(* PLC project ArfBot.project, CODESYS CODESYS V3.5 SP19 Patch 4 *)
(* stored: creationDateTime 2024-02-26T21:29:06.3801046, modificationDateTime 2024-02-26T21:28:27.7609543 *)

TYPE ST_CncCmd :
STRUCT
	StartPos: 		SMC_PosInfo;				
	OriConvention: 	SMC_ORI_CONVENTION:=SMC_ORI_CONVENTION.ZYX;
	Filename: 		STRING:='CNC_FromFile.cnc';
	CoordinateType: DUT_Command_CoordinateType:=DUT_Command_CoordinateType.Variable;
	ArrayIndex: 	INT:=GVL.DEC_START_POS;
	ArrayType: 		DUT_Command_ArrayType:=DUT_Command_ArrayType.StoredPosition;
END_STRUCT
END_TYPE

TYPE DUT_Command :
STRUCT
	CommandType: DUT_CommandType;
	CommandString: STRING(GVL.COMMAND_LEN);
END_STRUCT
END_TYPE

TYPE DUT_Program :
STRUCT
	ProgramName: STRING;
	Commands: ARRAY [GVL.PROG_CMDS_ARR_BEG..GVL.PROG_CMDS_ARR_END] OF DUT_Command;
END_STRUCT
END_TYPE

TYPE DUT_StoredPosition :
STRUCT
	Comment: STRING;
	Position: MC_COORD_REF;
END_STRUCT
END_TYPE

TYPE ST_VisionLocate :
STRUCT
    MaxParts: 		UINT:=1; // max number of parts to locate
    MaxOverlap: 	REAL:=0.0; // max overlap of parts. only needed if MaxParts is greater than zero.
    Score: 			REAL:=0.6; // min score
    ToleranceAngle: REAL:=90.0; // max angle +/- to search
	ResultPosition: UINT:=0; // location to store the results in the vision register array
	TemplateName: 	STRING:='Template.jpg'; // name of the template to search
	ScriptFilename: STRING:='FastTemplateMatching.py'; // name of the script that runs the vision program
END_STRUCT
END_TYPE

TYPE ST_VisionCalibrate :
STRUCT
    CheckerSize: REAL:=25.0; // this value is in user units ex mm
    CheckerXCount: UINT:=6; // count of checker blocks in x coordinate
    CheckerYCount: UINT:=9; // count of checker blocks in y coordinate
END_STRUCT
END_TYPE

TYPE ST_VisionCmd :
STRUCT
    CommandType: DUT_Command_VisionType;
    ImageWidth: UINT:=640; // pixel count in x direction (must be supported by camera)
    ImageHeight: UINT:=400; // pixel coutn in y direction (must be supported by camera)
    Calibrate: ST_VisionCalibrate;
    Locate: ST_VisionLocate;
	Timeout: UDINT:=60; // timeout in seconds
END_STRUCT
END_TYPE

TYPE DUT_VisionRegister EXTENDS DUT_StoredPosition :
STRUCT
	Scaling: REAL;
END_STRUCT
END_TYPE

TYPE DUT_Flags :
STRUCT
	Comment: STRING:='';
	Value: BOOL:=FALSE;
END_STRUCT
END_TYPE

TYPE ST_MoveCmd :
STRUCT
	// common
	MoveType: 					DUT_Command_MoveType:=DUT_Command_MoveType.DirectMove;
	Speed: 						LREAL:=0.0;
	CoordSystem: 				SMC_COORD_SYSTEM:=SMC_COORD_SYSTEM.ACS;
	
	// direct/linear moves
	PositionType: 				DUT_Command_PositionType:=DUT_Command_PositionType.AbsolutePosition;
	CoordinateType: 			DUT_Command_CoordinateType:=DUT_Command_CoordinateType.Literal;
	ArrayIndex: 				UINT:=0;
	ArrayType: 					DUT_Command_ArrayType:=DUT_Command_ArrayType.StoredPosition;
	CoordRef: 					MC_COORD_REF:=(X:=0, Y:=0, Z:=0, A:=0, B:=0, C:=0);
	
	// circular moves
	CircularCoordinateType: 	DUT_Command_CoordinateType:=DUT_Command_CoordinateType.Literal;
	CircularArrayIndex: 		UINT:=0;
	CircularArrayType: 			DUT_Command_ArrayType:=DUT_Command_ArrayType.StoredPosition;
	CircleMode: 				SMC_CIRC_MODE:=SMC_CIRC_MODE.CENTER;
	PathChoice: 				MC_CIRC_PATHCHOICE:=MC_CIRC_PATHCHOICE.CLOCKWISE;
	CoordRef2: 					MC_COORD_REF:=(X:=0, Y:=0, Z:=0, A:=0, B:=0, C:=0);
	
END_STRUCT
END_TYPE

TYPE ST_OutputCmd :
STRUCT
	OutputType: DUT_OutputType;
	OutputTarget: INT;
	OutputValue1: LREAL;
	OutputValue2: LREAL;
END_STRUCT
END_TYPE

TYPE ST_PauseCmd :
STRUCT
	PauseTime: TIME:=T#1S;
END_STRUCT
END_TYPE

TYPE ST_VarSetCmd :
STRUCT
	ArrayType: DUT_Command_ArrayType;
	ArrayIndex: INT;
	Coordinates: MC_COORD_REF;
END_STRUCT
END_TYPE

TYPE ST_LogicCmdIO :
STRUCT
	Input: ARRAY [GVL.DIG_IN_ARR_BEG..GVL.DIG_IN_ARR_END] OF BOOL;
	Output: ARRAY [GVL.DIG_OUT_ARR_BEG..GVL.DIG_OUT_ARR_END] OF BOOL;
	Register: ARRAY [GVL.REG_ARR_BEG..GVL.REG_ARR_END] OF UDINT;
	Counter: ARRAY [GVL.REG_ARR_BEG..GVL.REG_ARR_END] OF UDINT;
END_STRUCT
END_TYPE

TYPE ST_LogicCmd :
STRUCT
	IF_Condition : E_LogicIfCondition;
	IF_Condition_Idx: INT;
	IF_Condition_Operator: E_LogicIfConditionOperator;
	IF_Condition_Operator_Value: UDINT;
	THEN_Function: E_LogicFunction;
	THEN_Function_Value: UDINT;
	THEN_Function_Idx: INT;
	ELSE_Function: E_LogicFunction;
	ELSE_Function_Idx: INT;
	ELSE_Function_Value: UDINT;
END_STRUCT
END_TYPE

INTERFACE ITFModule
METHOD M_Start
VAR_INPUT
END_VAR
END_METHOD
METHOD M_Stop
VAR_INPUT
END_VAR
END_METHOD
METHOD M_Home
VAR_INPUT
END_VAR
END_METHOD
METHOD M_Abort
VAR_INPUT
END_VAR
END_METHOD
METHOD M_Hold
VAR_INPUT
END_VAR
END_METHOD
{attribute 'monitoring' := 'variable'}
PROPERTY PropCurrentState : PACK_ML.State
END_PROPERTY
{attribute 'monitoring' := 'variable'}
PROPERTY PropBusy : BOOL
END_PROPERTY
{attribute 'monitoring' := 'variable'}
PROPERTY PropError : BOOL
END_PROPERTY
{attribute 'monitoring' := 'variable'}
PROPERTY PropErrDescription : STRING
END_PROPERTY
END_INTERFACE

TYPE StringByteArray : UNION
  bArray : ARRAY[0..254] OF BYTE;
  sString : STRING(255);
END_UNION;
END_TYPE

PROGRAM _00_Main
VAR
	// drive parameters
	//SM_Drive_PosControl_J1.controller.fDeadTime := 2.0;
	//SM_Drive_PosControl_J2.controller.fDeadTime := 2.0;
	//SM_Drive_PosControl_J3.controller.fDeadTime := 2.0;
	//SM_Drive_PosControl_J4.controller.fDeadTime := 2.0;
	//SM_Drive_PosControl_J5.controller.fDeadTime := 2.0;
	//SM_Drive_PosControl_J6.controller.fDeadTime := 2.0;
	
	// homing
	SMC_Homing_J1,SMC_Homing_J2,SMC_Homing_J3: SMC_Homing;
	SMC_Homing_J4,SMC_Homing_J5,SMC_Homing_J6: SMC_Homing;
	HomingSequence: INT := 0;
	SMC_GroupPower_J: SMC_GroupPower;
	MC_GroupReset_J: MC_GroupReset;
	MC_GroupEnable_J : MC_GroupEnable;
	MC_GroupDisable_J : MC_GroupDisable;
	HomingVelocityFast: LREAL:= 20.0;
	HomingAcceleration: LREAL:= 100.0;
	
	// jogging
	ProcessJog: JogProcessor;
	JogStatusText: STRING(255);
	
	// cnc
	VisuStruct3DControl_J: VisuStruct3DControl;
	TrackPosition: PositionTracker;
	
	// command processor
	PowerOn: BOOL:=FALSE;
	_MoveCommandParser: ParseMoveCmd;
	ProcessMoveCommand: MoveCmdProcessor;
	ProcessMoveCommand_Execute: BOOL;
	ProcessMoveCommand_Reset: BOOL;
	ProcessMoveStatusText: STRING(255);
	ProcessCommands: CommandProcessor;
	ProcessCommands_Execute: BOOL;
	ProcessCommand_Cancel: BOOL;
	ProcessCommand_Reset: BOOL;
	ProcessCommand_ActiveProgram: UINT := 0;
	StMoveCmdPose1: ST_MoveCmd;
	StMoveCmdPose2: ST_MoveCmd;
	Abort: BOOL;
	
	// vision
	Vision_pResultRtrig: R_TRIG;
	Vision_BitmapVersion: INT;
	Vision_CaptureImage: BOOL;
	Vision_CapImgCmdAccepted: BOOL;
	Vision_RunCalibration: BOOL;
	Vision_RunCalCmdAccepted: BOOL;
	Vision_LocatePart: BOOL;
	Vision_LocPartCmdAccepted: BOOL;
	Vision_StreamCamera: BOOL;
	Vision_StrCamCmdAccepted: BOOL;
	Vision_Cancel: BOOL;
	Vision_Reset: BOOL;
	
	//
	BuildTests: BOOL:=FALSE;
	FirstScan: BOOL:=TRUE;

END_VAR

                    
{region "utility"}
		 
	IF FirstScan THEN
		A_Init();	
	END_IF
	
	IF BuildTests THEN
		BuildTests := FALSE;
		M_BuildTests();
	END_IF
	
{endregion}
     
{region "methods"}

    A_Jogging();
    A_Homing();
    A_CNC();
    A_Processor();
    A_Vision();
    
{endregion}

FirstScan:=FALSE;
                  

ACTION A_Homing:
                        IF NOT GVL.PowerOn AND HomingSequence > 0 AND HomingSequence < 999  THEN
	HomingSequence := 999;
END_IF

CASE HomingSequence OF
  999: //
		SMC_GroupPower_J.Enable := FALSE;
		SMC_GroupPower_J.bDriveStart := FALSE;
		SMC_GroupPower_J.bRegulatorOn := FALSE;
		MC_GroupEnable_J.Execute := FALSE;
		MC_GroupDisable_J.Execute := FALSE;
		ProcessMoveCommand_Execute := FALSE;
		SMC_Homing_J1.bExecute := FALSE;
		SMC_Homing_J2.bExecute := FALSE;
		SMC_Homing_J3.bExecute := FALSE;
		SMC_Homing_J4.bExecute := FALSE;
		SMC_Homing_J5.bExecute := FALSE;
		SMC_Homing_J6.bExecute := FALSE;
		SM_Drive_PosControl_J1.bSWLimitEnable := TRUE;
		SM_Drive_PosControl_J2.bSWLimitEnable := TRUE;
		SM_Drive_PosControl_J3.bSWLimitEnable := TRUE;
		SM_Drive_PosControl_J4.bSWLimitEnable := TRUE;
		SM_Drive_PosControl_J5.bSWLimitEnable := TRUE;
		SM_Drive_PosControl_J6.bSWLimitEnable := TRUE;
  		HomingSequence := 0;
		
	0: //
		IF GVL.Homing AND GVL.PowerOn THEN
			GVL.Homing := FALSE;
			SMC_GroupPower_J.Enable := TRUE;
			SMC_GroupPower_J.bDriveStart := TRUE;
			SMC_GroupPower_J.bRegulatorOn := TRUE;
			PersistentVars.Flags[GVL.HOME_COMPLETE].Value := FALSE;
			HomingSequence := 5;
		END_IF
		
	5:
		IF SMC_GroupPower_J.Status THEN
			MC_GroupEnable_J.Execute := TRUE;
			HomingSequence := 10;
		END_IF
		
	10:
		IF NOT MC_GroupEnable_J.Busy THEN
			HomingSequence := 20;
		END_IF
		
	20: //
		SMC_Homing_J1.bExecute := TRUE;
		SMC_Homing_J2.bExecute := TRUE;
		SMC_Homing_J3.bExecute := TRUE;
		SMC_Homing_J4.bExecute := TRUE;
		SMC_Homing_J5.bExecute := TRUE;
		SMC_Homing_J6.bExecute := TRUE;
		SMC_Homing_J1.bReturnToZero := FALSE;
		SMC_Homing_J2.bReturnToZero := FALSE;
		SMC_Homing_J3.bReturnToZero := FALSE;
		SMC_Homing_J4.bReturnToZero := FALSE;
		SMC_Homing_J5.bReturnToZero := FALSE;
		SMC_Homing_J6.bReturnToZero := FALSE;
		SMC_Homing_J1.fVelocitySlow := 10.0;
		SMC_Homing_J2.fVelocitySlow := 10.0;
		SMC_Homing_J3.fVelocitySlow := 10.0;
		SMC_Homing_J4.fVelocitySlow := 10.0;
		SMC_Homing_J5.fVelocitySlow := 10.0;
		SMC_Homing_J6.fVelocitySlow := 10.0;
		SM_Drive_PosControl_J1.bSWLimitEnable := FALSE;
		SM_Drive_PosControl_J2.bSWLimitEnable := FALSE;
		SM_Drive_PosControl_J3.bSWLimitEnable := FALSE;
		SM_Drive_PosControl_J4.bSWLimitEnable := FALSE;
		SM_Drive_PosControl_J5.bSWLimitEnable := FALSE;
		SM_Drive_PosControl_J6.bSWLimitEnable := FALSE;
		HomingSequence := 30;
		
	30: //
		IF SMC_Homing_J1.bDone
			AND SMC_Homing_J2.bDone
			AND SMC_Homing_J3.bDone
			AND SMC_Homing_J4.bDone
			AND SMC_Homing_J5.bDone
			AND SMC_Homing_J6.bDone THEN
				SMC_Homing_J1.bExecute := FALSE;
				SMC_Homing_J2.bExecute := FALSE;
				SMC_Homing_J3.bExecute := FALSE;
				SMC_Homing_J4.bExecute := FALSE;
				SMC_Homing_J5.bExecute := FALSE;
				SMC_Homing_J6.bExecute := FALSE;
				HomingSequence := 40;
		END_IF
		
	40: //
		SMC_Homing_J1.bExecute := TRUE;
		SMC_Homing_J2.bExecute := TRUE;
		SMC_Homing_J3.bExecute := TRUE;
		SMC_Homing_J4.bExecute := TRUE;
		SMC_Homing_J5.bExecute := TRUE;
		SMC_Homing_J6.bExecute := TRUE;
		IF NOT PersistentVars.Flags[GVL.HOM_TO_POSE_IDX].Value THEN
			SMC_Homing_J1.bReturnToZero := TRUE;
			SMC_Homing_J2.bReturnToZero := TRUE;
			SMC_Homing_J3.bReturnToZero := TRUE;
			SMC_Homing_J4.bReturnToZero := TRUE;
			SMC_Homing_J5.bReturnToZero := TRUE;
			SMC_Homing_J6.bReturnToZero := TRUE;
		END_IF
		SMC_Homing_J1.fVelocitySlow := 2.0;
		SMC_Homing_J2.fVelocitySlow := 2.0;
		SMC_Homing_J3.fVelocitySlow := 2.0;
		SMC_Homing_J4.fVelocitySlow := 2.0;
		SMC_Homing_J5.fVelocitySlow := 2.0;
		SMC_Homing_J6.fVelocitySlow := 2.0;
		HomingSequence := 50;
		
	50: //
		IF SMC_Homing_J1.bDone
			AND SMC_Homing_J2.bDone
			AND SMC_Homing_J3.bDone
			AND SMC_Homing_J4.bDone
			AND SMC_Homing_J5.bDone
			AND SMC_Homing_J6.bDone THEN
				SMC_Homing_J1.bExecute := FALSE;
				SMC_Homing_J2.bExecute := FALSE;
				SMC_Homing_J3.bExecute := FALSE;
				SMC_Homing_J4.bExecute := FALSE;
				SMC_Homing_J5.bExecute := FALSE;
				SMC_Homing_J6.bExecute := FALSE;
				IF NOT PersistentVars.Flags[GVL.HOM_TO_POSE_IDX].Value THEN
					HomingSequence := 60;
				ELSE
					HomingSequence := 100;
				END_IF
				PersistentVars.Flags[GVL.HOME_COMPLETE].Value := TRUE;
		END_IF
		
	60:
		MC_GroupDisable_J.Execute := TRUE;
		HomingSequence := 70;
		
	70:
		IF NOT MC_GroupDisable_J.Busy THEN
			HomingSequence := 999;
		END_IF
		
	100: //
		ProcessMoveCommand.Command := GVL.Pose2;
		ProcessMoveCommand.M_Start();
		HomingSequence := 110;
		
	110: //
		IF ProcessMoveCommand.ItfUnitMode.CurrentState = PACK_ML.State.Idle 
			OR NOT ProcessMoveCommand_Execute THEN
				ProcessMoveCommand_Execute := FALSE;
				HomingSequence := 999;
		END_IF

END_CASE

SMC_Homing_J1(
	Axis:=SM_Drive_PosControl_J1 , 
	bExecute:= ,
	fHomePosition:= PersistentVars.StoredPositions[GVL.HOM_POS_IDX].Position.X, 
	fVelocitySlow:= , 
	fVelocityFast:= HomingVelocityFast, 
	fAcceleration:= HomingAcceleration, 
	fDeceleration:= HomingAcceleration, 
	fJerk:= 1000.0, 
	nDirection:= MC_direction.negative, 
	bReferenceSwitch:= NOT _10_Drives.rx_j1_limit, 
	fSignalDelay:= , 
	nHomingMode:= , 
	bReturnToZero:= , 
	bIndexOccured:= , 
	fIndexPosition:= , 
	bIgnoreHWLimit:= TRUE, 
	bDone=> , 
	bBusy=> , 
	bCommandAborted=> , 
	bError=> , 
	nErrorID=> , 
	bStartLatchingIndex=> );
	
SMC_Homing_J2(
	Axis:=SM_Drive_PosControl_J2 , 
	bExecute:= , 
	fHomePosition:= PersistentVars.StoredPositions[GVL.HOM_POS_IDX].Position.Y,  
	fVelocitySlow:= , 
	fVelocityFast:= HomingVelocityFast, 
	fAcceleration:= HomingAcceleration, 
	fDeceleration:= HomingAcceleration,
	fJerk:= 1000.0, 
	nDirection:= MC_Direction.negative, 
	bReferenceSwitch:= NOT _10_Drives.rx_j2_limit, 
	fSignalDelay:= , 
	nHomingMode:= , 
	bReturnToZero:= , 
	bIndexOccured:= , 
	fIndexPosition:= , 
	bIgnoreHWLimit:= TRUE, 
	bDone=> , 
	bBusy=> , 
	bCommandAborted=> , 
	bError=> , 
	nErrorID=> , 
	bStartLatchingIndex=> );
	
SMC_Homing_J3(
	Axis:=SM_Drive_PosControl_J3 , 
	bExecute:= , 
	fHomePosition:= PersistentVars.StoredPositions[GVL.HOM_POS_IDX].Position.Z, 
	fVelocitySlow:= , 
	fVelocityFast:= HomingVelocityFast, 
	fAcceleration:= HomingAcceleration, 
	fDeceleration:= HomingAcceleration,
	fJerk:= 1000.0, 
	nDirection:= MC_Direction.positive, 
	bReferenceSwitch:= NOT _10_Drives.rx_j3_limit, 
	fSignalDelay:= , 
	nHomingMode:= , 
	bReturnToZero:= , 
	bIndexOccured:= , 
	fIndexPosition:= , 
	bIgnoreHWLimit:= TRUE, 
	bDone=> , 
	bBusy=> , 
	bCommandAborted=> , 
	bError=> , 
	nErrorID=> , 
	bStartLatchingIndex=> );
	
SMC_Homing_J4(
	Axis:=SM_Drive_PosControl_J4 , 
	bExecute:= ,
	fHomePosition:= PersistentVars.StoredPositions[GVL.HOM_POS_IDX].Position.A, 
	fVelocitySlow:= , 
	fVelocityFast:= HomingVelocityFast, 
	fAcceleration:= HomingAcceleration, 
	fDeceleration:= HomingAcceleration,
	fJerk:= 1000.0, 
	nDirection:= MC_Direction.positive, 
	bReferenceSwitch:= NOT _10_Drives.rx_j4_limit, 
	fSignalDelay:= , 
	nHomingMode:= , 
	bReturnToZero:= , 
	bIndexOccured:= , 
	fIndexPosition:= , 
	bIgnoreHWLimit:= TRUE, 
	bDone=> , 
	bBusy=> , 
	bCommandAborted=> , 
	bError=> , 
	nErrorID=> , 
	bStartLatchingIndex=> );
	
SMC_Homing_J5(
	Axis:=SM_Drive_PosControl_J5 , 
	bExecute:= , 
	fHomePosition:= PersistentVars.StoredPositions[GVL.HOM_POS_IDX].Position.B,  
	fVelocitySlow:= , 
	fVelocityFast:= HomingVelocityFast, 
	fAcceleration:= HomingAcceleration, 
	fDeceleration:= HomingAcceleration,
	fJerk:= 1000, 
	nDirection:= MC_Direction.positive, 
	bReferenceSwitch:= NOT _10_Drives.rx_j5_limit, 
	fSignalDelay:= , 
	nHomingMode:= , 
	bReturnToZero:= , 
	bIndexOccured:= , 
	fIndexPosition:= , 
	bIgnoreHWLimit:= TRUE, 
	bDone=> , 
	bBusy=> , 
	bCommandAborted=> , 
	bError=> , 
	nErrorID=> , 
	bStartLatchingIndex=> );
	
SMC_Homing_J6(
	Axis:=SM_Drive_PosControl_J6 , 
	bExecute:= , 
	fHomePosition:= PersistentVars.StoredPositions[GVL.HOM_POS_IDX].Position.C, 
	fVelocitySlow:= , 
	fVelocityFast:= HomingVelocityFast, 
	fAcceleration:= HomingAcceleration, 
	fDeceleration:= HomingAcceleration,
	fJerk:= 1000.0, 
	nDirection:= MC_Direction.negative, 
	bReferenceSwitch:= NOT _10_Drives.rx_j6_limit, 
	fSignalDelay:= , 
	nHomingMode:= , 
	bReturnToZero:= , 
	bIndexOccured:= , 
	fIndexPosition:= , 
	bIgnoreHWLimit:= TRUE, 
	bDone=> , 
	bBusy=> , 
	bCommandAborted=> , 
	bError=> , 
	nErrorID=> , 
	bStartLatchingIndex=> );

SMC_GroupPower_J(
	AxisGroup:= ArfBotAxisGroup, 
	Enable:=,
	bRegulatorOn:= SMC_GroupPower_J.Enable,
	bDriveStart:= SMC_GroupPower_J.Enable, 
	Status=> , 
	Busy=> , 
	Error=> , 
	ErrorID=> );
		 
MC_GroupEnable_J(
	AxisGroup:=ArfBotAxisGroup,
	Execute:=,
	CompatibilityOptions:=,
	Done=>,
	Busy=>,
	Error=>,
	ErrorID=>);
		 
MC_GroupDisable_J(
	AxisGroup:=ArfBotAxisGroup,
	Execute:=,
	Done=>,
	Busy=>,
	Error=>,
	ErrorID=>);	
		 
MC_GroupReset_J(
	AxisGroup:=ArfBotAxisGroup , 
	Execute:= GVL.Reset, 
	Done=> , 
	Busy=> , 
	Error=> , 
	ErrorID=> );
                      
END_ACTION

ACTION A_Processor:
                        
//	TODO need to get this removed and instead build a program for the poses
IF GVL.MoveToPose1 THEN
	GVL.MoveToPose1 := FALSE;
	IF GVL.PowerOn AND PersistentVars.Flags[GVL.HOME_COMPLETE].Value THEN
		ProcessMoveCommand.Command := GVL.Pose1;
		ProcessMoveCommand.M_Start();
	END_IF
ELSIF GVL.MoveToPose2 THEN
	GVL.MoveToPose2 := FALSE;
	IF GVL.PowerOn AND PersistentVars.Flags[GVL.HOME_COMPLETE].Value THEN
		ProcessMoveCommand.Command := GVL.Pose2;
		ProcessMoveCommand.M_Start();
	END_IF
END_IF

// TODO need to get this removed and instead build a program for the poses
ProcessMoveCommand(
	StoredPositions:= PersistentVars.StoredPositions,
	VisionRegisters:= PersistentVars.VisionRegisters,
	Flags:= PersistentVars.Flags,
	AxisGroup:= ArfBotAxisGroup, 
	Acceleration:= 1000, 
	AccFactor:= 0.05,
	Jerk:= 1000,
	JerkFactor:= 1, 
	Position=> ,
	ItfUnitMode=> , 
	Error=> );
IF ProcessMoveCommand_Reset OR GVL.Reset THEN
	ProcessMoveCommand_Reset := FALSE;
	ProcessMoveStatusText := '';
	ProcessMoveCommand.M_Home();
END_IF
IF ProcessMoveCommand.Error THEN
	ProcessMoveStatusText := CONCAT('Move Processor Error: ',ProcessMoveCommand.ErrorDescription) ;
END_IF

//
IF Abort THEN
	Abort := FALSE;
	IF NOT GVL.PowerOn THEN
		ProcessCommands.M_Abort();
		ProcessMoveCommand.M_Abort();
	END_IF
END_IF
IF ProcessCommands_Execute THEN
	ProcessCommands_Execute := FALSE;
	ProcessCommands.Commands := PersistentVars.Programs[ProcessCommand_ActiveProgram].Commands;
	ProcessCommands.M_Start();
END_IF
IF ProcessCommand_Cancel THEN
	ProcessCommand_Cancel := FALSE;
	ProcessCommands.M_Stop();
END_IF
IF ProcessCommand_Reset OR GVL.Reset THEN
	ProcessCommand_Reset := FALSE;
	ProcessCommands.M_Home();
END_IF
ProcessCommands(
	StoredPositions:=PersistentVars.StoredPositions,
	VisionRegisters:=PersistentVars.VisionRegisters,
	Flags:=PersistentVars.Flags,
	AxisGroup:= ArfBotAxisGroup,
	Servo1:= AdafruitPwm01,
	Servo2:= AdafruitPwm02,
	Enable:= GVL.PowerOn AND PersistentVars.Flags[GVL.HOME_COMPLETE].Value,
	Commands:= , 
	ActiveCommand => ,
	Error=> ,
	StatusText=>);	
                      
END_ACTION

ACTION A_CNC:
                        
// track position of robot end effector to display on hmi
TrackPosition(
	AxisGroup:=ArfBotAxisGroup,
	SM3_Drive_PosControl_J1:=SM_Drive_PosControl_J1,
	SM3_Drive_PosControl_J2:=SM_Drive_PosControl_J2,
	SM3_Drive_PosControl_J3:=SM_Drive_PosControl_J3,
	SM3_Drive_PosControl_J4:=SM_Drive_PosControl_J4,
	SM3_Drive_PosControl_J5:=SM_Drive_PosControl_J5,
	SM3_Drive_PosControl_J6:=SM_Drive_PosControl_J6,
	VisuStruct3DTrack=>,
	Arm=>,
	Elbow=>,
	Hand=>);
	
(*ProcessCnc(
	AxisGroup:=ArfBotAxisGroup,
	SM3_Drive_PosControl_J1:=SM_Drive_PosControl_J1,
	SM3_Drive_PosControl_J2:=SM_Drive_PosControl_J2,
	SM3_Drive_PosControl_J3:=SM_Drive_PosControl_J3,
	SM3_Drive_PosControl_J4:=SM_Drive_PosControl_J4,
	SM3_Drive_PosControl_J5:=SM_Drive_PosControl_J5,
	SM3_Drive_PosControl_J6:=SM_Drive_PosControl_J6,
	GapVelocity:= , 
	AvoidGaps:= , 
	GapAccel:= );*)

// set the start position for the MC_NCDecoder
// alternatively, we can set this in the CNC program properties
(*GVL.StartPos.dX:=PersistentVars.StoredPositions[GVL.DEC_START_POS].Position.X;
GVL.StartPos.dY:=PersistentVars.StoredPositions[GVL.DEC_START_POS].Position.Y;
GVL.StartPos.dZ:=PersistentVars.StoredPositions[GVL.DEC_START_POS].Position.Z;
GVL.StartPos.dA:=PersistentVars.StoredPositions[GVL.DEC_START_POS].Position.A;
GVL.StartPos.dB:=PersistentVars.StoredPositions[GVL.DEC_START_POS].Position.B;
GVL.StartPos.dC:=PersistentVars.StoredPositions[GVL.DEC_START_POS].Position.C;

IF TestExecute THEN
	TestExecute := FALSE;
	ProcessCnc.M_Execute(	FileName:='CNC_FromFile.cnc', 
							StartPos:=GVL.StartPos); // TODO 
END_IF
IF TestReset THEN
	TestReset := FALSE;
	ProcessCnc.M_Reset();
END_IF
IF TestCancel THEN
	TestCancel := FALSE;
	ProcessCnc.M_Cancel();
END_IF*)
                      
END_ACTION

ACTION A_Jogging:
                        
ProcessJog(
	AxisGroup:= ArfBotAxisGroup,
	Enable:= GVL.PowerOn,
	Reset:= GVL.Reset,
	ABC_as_ACS=>,
	CoordSystem=>, 
	Position=>, 
	Done=> , 
	Busy=> , 
	Error=> , 
	ErrorID=> );
IF ProcessJog.Reset THEN
	JogStatusText := '';
END_IF
IF ProcessJog.Error THEN
	JogStatusText := CONCAT('Jog Processor Error: ',
						CONCAT(TO_STRING(ProcessJog.ErrorID),
						CONCAT(' ', SMC_ErrorString(ProcessJog.ErrorID,
									SMC_Language_Type.english)))) ;
END_IF

                      
END_ACTION

ACTION A_Vision:
                        
// tell HMI to update image
//Vision_pResultRtrig(clk := _40_Vision.ProcessVisionCommand.ItfUnitMode.CurrentState = PACK_ML.State.Idle); TODO this causes an exception because ProcessVisionCommand has not went through first scan yet
Vision_pResultRtrig(clk := NOT _40_Vision.ProcessVisionCommand.Busy);
IF Vision_pResultRtrig.Q THEN
	Vision_BitmapVersion := Vision_BitmapVersion + 1;
END_IF

                      
END_ACTION

ACTION A_Init:
                        
// check if arfbot has been initialized
IF NOT PersistentVars.Flags[GVL.INIT_POS_IDX].Value THEN
	// poses
	PersistentVars.Flags[GVL.HOM_TO_POSE_IDX].Value := FALSE;
	PersistentVars.StoredPositions[GVL.POSE_1_IDX].Position.X := 0.0;
	PersistentVars.StoredPositions[GVL.POSE_1_IDX].Position.Y := 0.0;
	PersistentVars.StoredPositions[GVL.POSE_1_IDX].Position.Z := -30.0;
	PersistentVars.StoredPositions[GVL.POSE_1_IDX].Position.A := 0.0;
	PersistentVars.StoredPositions[GVL.POSE_1_IDX].Position.B := -30.0;
	PersistentVars.StoredPositions[GVL.POSE_1_IDX].Position.C := 0.0;
	PersistentVars.StoredPositions[GVL.POSE_2_IDX].Position.X := 0.0;
	PersistentVars.StoredPositions[GVL.POSE_2_IDX].Position.Y := 30.0;
	PersistentVars.StoredPositions[GVL.POSE_2_IDX].Position.Z := -30.0;
	PersistentVars.StoredPositions[GVL.POSE_2_IDX].Position.A := 0.0;
	PersistentVars.StoredPositions[GVL.POSE_2_IDX].Position.B := 30.0;
	PersistentVars.StoredPositions[GVL.POSE_2_IDX].Position.C := 0.0;
		 
	// decoder
	PersistentVars.StoredPositions[GVL.DEC_START_POS].Position.X := 300.0; // TODO need to verify all 6 of these
	PersistentVars.StoredPositions[GVL.DEC_START_POS].Position.Y := 0.0;
	PersistentVars.StoredPositions[GVL.DEC_START_POS].Position.Z := -400.0;
	PersistentVars.StoredPositions[GVL.DEC_START_POS].Position.A := 0.0;
	PersistentVars.StoredPositions[GVL.DEC_START_POS].Position.B := 0.0;
	PersistentVars.StoredPositions[GVL.DEC_START_POS].Position.C := 0.0;
		 
	
	// set homing offsets
	PersistentVars.StoredPositions[GVL.HOM_POS_IDX].Position.X := 167.0; // J1 initial home offset
	PersistentVars.StoredPositions[GVL.HOM_POS_IDX].Position.Y := 42.41; // J2 initial home offset
	PersistentVars.StoredPositions[GVL.HOM_POS_IDX].Position.Z := -57.35; // J3 initial home offset
	PersistentVars.StoredPositions[GVL.HOM_POS_IDX].Position.A := -169.66; // J4 initial home offset
	PersistentVars.StoredPositions[GVL.HOM_POS_IDX].Position.B := -94.106; // J5 initial home offset
	PersistentVars.StoredPositions[GVL.HOM_POS_IDX].Position.C := 171.581; // J6 initial home offset
	
	//
	M_BuildTests();
		 
	// indicate initialized
	PersistentVars.Flags[GVL.INIT_POS_IDX].Value := TRUE;
END_IF

// 
PersistentVars.StoredPositions[GVL.HOM_POS_IDX].Comment := 'Home Offsets J1, J2, J3, J4, J5, J6';
PersistentVars.StoredPositions[GVL.DEC_START_POS].Comment := 'NC Decoder Start Position';
PersistentVars.StoredPositions[GVL.TCP_POS_IDX].Comment := 'TCP Offset';
PersistentVars.StoredPositions[GVL.PC2_POS_IDX].Comment := 'PCS 2 Offset';
PersistentVars.StoredPositions[GVL.PC1_POS_IDX].Comment := 'PCS 1 Offset';
PersistentVars.StoredPositions[GVL.MCS_POS_IDX].Comment := 'MCS Offset';

//	 
PersistentVars.StoredPositions[GVL.POSE_1_IDX].Comment := 'Pose 1 coordinates';
PersistentVars.StoredPositions[GVL.POSE_2_IDX].Comment := 'Pose 2 coordinates';
PersistentVars.StoredPositions[GVL.POSE_3_IDX].Comment := 'Pose 3 coordinates';
PersistentVars.StoredPositions[GVL.POSE_4_IDX].Comment := 'Pose 4 coordinates';
PersistentVars.StoredPositions[GVL.POSE_5_IDX].Comment := 'Pose 5 coordinates';

//
PersistentVars.Flags[GVL.HOM_TO_POSE_IDX].Comment := 'Finish home at Pose';

//
PersistentVars.Flags[GVL.HOME_COMPLETE].Comment := 'Indicates all axes are homed';
PersistentVars.Flags[GVL.HOME_COMPLETE].Value := FALSE;

// build pose commands
//
StMoveCmdPose1.MoveType 		:= DUT_Command_MoveType.DirectMove;
StMoveCmdPose1.PositionType 	:= DUT_Command_PositionType.AbsolutePosition;
StMoveCmdPose1.CoordinateType 	:= DUT_Command_CoordinateType.Literal;
StMoveCmdPose1.Speed 			:= 20;
StMoveCmdPose1.CoordSystem 		:= SMC_COORD_SYSTEM.ACS;
StMoveCmdPose1.CoordRef 		:= PersistentVars.StoredPositions[GVL.POSE_1_IDX].Position;
GVL.Pose1 := BuildMoveCmd(StMoveCmdPose1);
//
StMoveCmdPose2.MoveType 		:= DUT_Command_MoveType.DirectMove;
StMoveCmdPose2.PositionType 	:= DUT_Command_PositionType.AbsolutePosition;
StMoveCmdPose2.CoordinateType 	:= DUT_Command_CoordinateType.Literal;
StMoveCmdPose2.Speed 			:= 20;
StMoveCmdPose2.CoordSystem 		:= SMC_COORD_SYSTEM.ACS;
StMoveCmdPose2.CoordRef 		:= PersistentVars.StoredPositions[GVL.POSE_2_IDX].Position;
GVL.Pose2 := BuildMoveCmd(StMoveCmdPose2);
                      
END_ACTION

METHOD M_BuildTests
VAR_INPUT
END_VAR
VAR
	_i, _j, _k: INT;
END_VAR
                          
//
FOR _i := GVL.PROG_CMDS_ARR_BEG TO GVL.PROG_CMDS_ARR_END BY 1 DO
	PersistentVars.Programs[1].Commands[_i].CommandType := DUT_CommandType.Disabled;
	PersistentVars.Programs[1].Commands[_i].CommandString := '';
END_FOR
PersistentVars.Programs[1].ProgramName := 'Vision Pick and Place';
PersistentVars.Programs[1].Commands[0].CommandType := DUT_CommandType.VarSetCommand;
PersistentVars.Programs[1].Commands[0].CommandString := 'STO 0046 +0000.00 +0000.00 +0000.00 +0090.00 +0000.00 +0000.00';
PersistentVars.Programs[1].Commands[1].CommandType := DUT_CommandType.MoveCommand;
PersistentVars.Programs[1].Commands[1].CommandString := 'DIR ABS 020 ACS LIT 00000.00 00030.00 -0030.00 00000.00 00030.00 00000.00';
PersistentVars.Programs[1].Commands[2].CommandType := DUT_CommandType.OutputCommand;
PersistentVars.Programs[1].Commands[2].CommandString := 'DIG 1 1';
PersistentVars.Programs[1].Commands[3].CommandType := DUT_CommandType.VisionCommand;
PersistentVars.Programs[1].Commands[3].CommandString := 'LOC 640 400 0060 001 000.0 0.8 030.0 000 Template.jpg FastTemplateMatching.py';
PersistentVars.Programs[1].Commands[4].CommandType := DUT_CommandType.OutputCommand;
PersistentVars.Programs[1].Commands[4].CommandString := 'DIG 1 0';
PersistentVars.Programs[1].Commands[5].CommandType := DUT_CommandType.MoveCommand;
PersistentVars.Programs[1].Commands[5].CommandString := 'DIR ABS 050 PC1 LIT 00000.00 00000.00 -0010.00 00000.00 00000.00 00000.00';
PersistentVars.Programs[1].Commands[6].CommandType := DUT_CommandType.MoveCommand;
PersistentVars.Programs[1].Commands[6].CommandString := 'DIR ABS 050 PC1 VAR VIS 000';
PersistentVars.Programs[1].Commands[7].CommandType := DUT_CommandType.OutputCommand;
PersistentVars.Programs[1].Commands[7].CommandString := 'SRV 1 30.0 360.0';
PersistentVars.Programs[1].Commands[8].CommandType := DUT_CommandType.MoveCommand;
PersistentVars.Programs[1].Commands[8].CommandString := 'LIN REL 050 TCS LIT 00000.00 00000.00 00010.00 00000.00 00000.00 00000.00';
PersistentVars.Programs[1].Commands[9].CommandType := DUT_CommandType.OutputCommand;
PersistentVars.Programs[1].Commands[9].CommandString := 'SRV 1 0.0 360.0';
PersistentVars.Programs[1].Commands[10].CommandType := DUT_CommandType.PauseCommand;
PersistentVars.Programs[1].Commands[10].CommandString := 'T#1s';
PersistentVars.Programs[1].Commands[11].CommandType := DUT_CommandType.MoveCommand;
PersistentVars.Programs[1].Commands[11].CommandString := 'LIN REL 050 TCS LIT 00000.00 00000.00 -0010.00 00000.00 00000.00 00000.00';
PersistentVars.Programs[1].Commands[12].CommandType := DUT_CommandType.MoveCommand;
PersistentVars.Programs[1].Commands[12].CommandString := 'DIR ABS 050 PC1 LIT 00000.00 00000.00 -0050.00 00000.00 00000.00 00000.00';
PersistentVars.Programs[1].Commands[13].CommandType := DUT_CommandType.OutputCommand;
PersistentVars.Programs[1].Commands[13].CommandString := 'SRV 1 30.0 360.0';

//
FOR _i := GVL.PROG_CMDS_ARR_BEG TO GVL.PROG_CMDS_ARR_END BY 1 DO
	PersistentVars.Programs[2].Commands[_i].CommandType := DUT_CommandType.Disabled;
	PersistentVars.Programs[2].Commands[_i].CommandString := '';
END_FOR
PersistentVars.Programs[2].ProgramName := 'PCS1 Corners';
PersistentVars.Programs[2].Commands[0].CommandType := DUT_CommandType.VarSetCommand;
PersistentVars.Programs[2].Commands[0].CommandString := 'STO 0046 +0000.00 +0000.00 +0000.00 +0090.00 +0000.00 +0000.00';
PersistentVars.Programs[2].Commands[1].CommandType := DUT_CommandType.MoveCommand;
PersistentVars.Programs[2].Commands[1].CommandString := 'DIR ABS 050 PC1 LIT 0 0 0 0 0 0';
PersistentVars.Programs[2].Commands[2].CommandType := DUT_CommandType.MoveCommand;
PersistentVars.Programs[2].Commands[2].CommandString := 'LIN REL 100 TCS LIT 0.0 200.0 0.0 0.0 0.0 0.0';
PersistentVars.Programs[2].Commands[3].CommandType := DUT_CommandType.MoveCommand;
PersistentVars.Programs[2].Commands[3].CommandString := 'LIN REL 100 TCS LIT 00125.00 00000.00 00000.00 00000.00 00000.00 00000.00';
PersistentVars.Programs[2].Commands[4].CommandType := DUT_CommandType.MoveCommand;
PersistentVars.Programs[2].Commands[4].CommandString := 'LIN REL 100 TCS LIT 00000.00 -0200.00 00000.00 00000.00 00000.00 00000.00';
PersistentVars.Programs[2].Commands[5].CommandType := DUT_CommandType.MoveCommand;
PersistentVars.Programs[2].Commands[5].CommandString := 'LIN REL 100 TCS LIT -0125.00 00000.00 00000.00 00000.00 00000.00 00000.00';
PersistentVars.Programs[2].Commands[6].CommandType := DUT_CommandType.MoveCommand;
PersistentVars.Programs[2].Commands[6].CommandString := 'DIR ABS 050 ACS LIT +00 +30 -30 +00 +30 +00';

//
FOR _i := GVL.PROG_CMDS_ARR_BEG TO GVL.PROG_CMDS_ARR_END BY 1 DO
	PersistentVars.Programs[3].Commands[_i].CommandType := DUT_CommandType.Disabled;
	PersistentVars.Programs[3].Commands[_i].CommandString := '';
END_FOR
PersistentVars.Programs[3].ProgramName := 'Cnc Validation';
PersistentVars.Programs[3].Commands[0].CommandType := DUT_CommandType.CncCommand;
PersistentVars.Programs[3].Commands[0].CommandString := 'CNC_FromFile.cnc XYZ VAR STO 45';
PersistentVars.Programs[3].Commands[1].CommandType := DUT_CommandType.CncCommand;
PersistentVars.Programs[3].Commands[1].CommandString := 'CNC_FromFile.cnc XYZ LIT +0300.00 +0000.00 -0300.00 +0000.00 +0000.00 +0000.00';

//
FOR _i := GVL.PROG_CMDS_ARR_BEG TO GVL.PROG_CMDS_ARR_END BY 1 DO
	PersistentVars.Programs[4].Commands[_i].CommandType := DUT_CommandType.Disabled;
	PersistentVars.Programs[4].Commands[_i].CommandString := '';
END_FOR
PersistentVars.Programs[4].ProgramName := 'Vision Validation';
PersistentVars.Programs[4].Commands[0].CommandType := DUT_CommandType.VisionCommand;
PersistentVars.Programs[4].Commands[0].CommandString := 'LOC 640 400 60 1 0.0 0.8 30.0 10 Template.jpg FastTemplateMatching.py';
PersistentVars.Programs[4].Commands[1].CommandType := DUT_CommandType.VisionCommand;
PersistentVars.Programs[4].Commands[1].CommandString := 'LOC 640 400 60 1 0.0 0.8 30.0 4 strippers2.jpg FastTemplateMatching.py';

//
FOR _i := GVL.PROG_CMDS_ARR_BEG TO GVL.PROG_CMDS_ARR_END BY 1 DO
	PersistentVars.Programs[5].Commands[_i].CommandType := DUT_CommandType.Disabled;
	PersistentVars.Programs[5].Commands[_i].CommandString := '';
END_FOR
PersistentVars.Programs[5].ProgramName := 'VarSet Validation';
PersistentVars.Programs[5].Commands[0].CommandType := DUT_CommandType.VarSetCommand;
PersistentVars.Programs[5].Commands[0].CommandString := 'STO 1 6.0 5.0 4.0 3.0 2.0 1.0 ';
PersistentVars.Programs[5].Commands[1].CommandType := DUT_CommandType.VarSetCommand;
PersistentVars.Programs[5].Commands[1].CommandString := 'VIS 2 1 2 3 4 5 6';
PersistentVars.Programs[5].Commands[2].CommandType := DUT_CommandType.VarSetCommand;
PersistentVars.Programs[5].Commands[2].CommandString := 'FLG 3 1';


//
FOR _i := GVL.PROG_CMDS_ARR_BEG TO GVL.PROG_CMDS_ARR_END BY 1 DO
	PersistentVars.Programs[6].Commands[_i].CommandType := DUT_CommandType.Disabled;
	PersistentVars.Programs[6].Commands[_i].CommandString := '';
END_FOR
PersistentVars.Programs[6].ProgramName := 'Logic Validation';
PersistentVars.Programs[6].Commands[0].CommandType := DUT_CommandType.LogicCommand;
PersistentVars.Programs[6].Commands[0].CommandString := 'IF INPUT 1 EQU 1 THEN OUTPUT 1 1 ELSE OUTPUT 1 0';
PersistentVars.Programs[6].Commands[1].CommandType := DUT_CommandType.LogicCommand;
PersistentVars.Programs[6].Commands[1].CommandString := 'IF INPUT 1 EQU 1 THEN CNTUP 1 ELSE CNTUP 2';
PersistentVars.Programs[6].Commands[2].CommandType := DUT_CommandType.LogicCommand;
PersistentVars.Programs[6].Commands[2].CommandString := 'IF COUNTER 2 GRE 10 THEN NOP ELSE JUMP 0';
















                        
END_METHOD
END_PROGRAM

PROGRAM _10_Drives
VAR	
	SetVelocity: ARRAY [0..5] OF REAL;
	EncPosition: ARRAY [0..5] OF DINT;
	
	bufferIdx: INT;
	jointIdx: INT;
	
	HeartbeatOn: TON;
	HeartbeatOff: TON;
	HeartbeatPt: TIME:=T#1000MS;
	SysLTime, SysLTimeLast: LTIME;
	TransferTime: LTIME:=LTIME#100US;
	TransferTrigger: BOOL;
	
	pabyTxBuffer: ARRAY [0..31] OF BYTE;
	pabyRxBuffer: ARRAY [0..31] OF BYTE;
	
	transferlentx: UDINT:=32;
	transferlenrx: UDINT:=32;
	i2caddress: USINT:=8;
	
	rx_heartbeat: BOOL;
	rx_en, tx_en: BOOL;
	rx_alarm: BOOL;
	rx_heartbeat_lost: BOOL;
	rx_j1_limit, rx_j2_limit, rx_j3_limit: BOOL;
	rx_j4_limit, rx_j5_limit, rx_j6_limit: BOOL;
	
	
	
	
	
	
	TestMove_J6:BOOL;
	PosStart1_J6: DINT;
	PosStart2_J6: DINT;
	PosEnd1_J6: DINT;
	PosEnd2_J6: DINT;
	TestMoveWaitTimer: TON;
	TestMoveWaitTimerPT: TIME:=T#2S;
	
	TestMoveStep: INT;
	
END_VAR

                    
HeartbeatOn(in:=NOT HeartbeatOff.Q,PT:=HeartbeatPt);
HeartbeatOff(in:=HeartbeatOn.Q,PT:=HeartbeatPt);

// need to use system time to transfer faster than 1ms
SysLTime := LTIME();
IF SysLTime - SysLTimeLast > TransferTime THEN
	SysLTimeLast := SysLTime;
	TransferTrigger := NOT TransferTrigger;
END_IF

// handle outputs
// index 0 is for system outputs
pabyTxBuffer[0].0:=HeartbeatOn.Q; 	// heartbeat
pabyTxBuffer[0].1:=tx_en; 			// enable drives
//pabyTxBuffer[0].2:=GVL.Homing;		// homing sts
// pabyTxBuffer[0].3:=; //
// pabyTxBuffer[0].4:=; //
// pabyTxBuffer[0].5:=; //
// pabyTxBuffer[0].6:=; //
// pabyTxBuffer[0].7:=; //

// index 1 through 24 is for velocity to drive
bufferIdx := 1;
FOR jointIdx := 0 TO 5 BY 1 DO
	MEMUtils.MemCpy(pbyDest:=ADR(pabyTxBuffer[bufferIdx]), 
					pbySrc:=ADR(SetVelocity[jointIdx]), 
					dwSize:=SIZEOF(SetVelocity[jointIdx]));
	bufferIdx := bufferIdx + 4;
END_FOR
//pabyTxBuffer[25]:=;
//pabyTxBuffer[26]:=;
//pabyTxBuffer[27]:=;
//pabyTxBuffer[28]:=;
//pabyTxBuffer[29]:=;
//pabyTxBuffer[30]:=;

// index 31 will be for gpio byte (bits 0 through 7)
pabyTxBuffer[31].0 := GVL.DigitalOutput[0];
pabyTxBuffer[31].1 := GVL.DigitalOutput[1];
pabyTxBuffer[31].2 := GVL.DigitalOutput[2];
pabyTxBuffer[31].3 := GVL.DigitalOutput[3];
pabyTxBuffer[31].4 := GVL.DigitalOutput[4];
pabyTxBuffer[31].5 := GVL.DigitalOutput[5];
pabyTxBuffer[31].6 := GVL.DigitalOutput[6];
pabyTxBuffer[31].7 := GVL.DigitalOutput[7];

// read and write to drive
IF TransferTrigger THEN
	I2C_master.write(usiAddress:=i2caddress,
					pbyBuffer:=ADR(pabyTxBuffer),
					nBufferLen:=transferlentx);
	I2C_master.read(usiAddress:=i2caddress,
					pbyBuffer:=ADR(pabyRxBuffer),
					nBufferLen:=transferlenrx);
END_IF

// handle inputs
// index 0 is for system inputs
rx_heartbeat 		:= pabyRxBuffer[0].0;
rx_en 				:= pabyRxBuffer[0].1;
rx_alarm 			:= pabyRxBuffer[0].2;
//rx_ 				:= pabyRxBuffer[0].3;
//rx_ 				:= pabyRxBuffer[0].4;
//rx_ 				:= pabyRxBuffer[0].5;
//rx_ 				:= pabyRxBuffer[0].6;
rx_heartbeat_lost 	:= pabyRxBuffer[0].7;

// index 1 through 24 is for encoder data from drive
bufferIdx := 1;
FOR jointIdx := 0 TO 5 BY 1 DO
	MEMUtils.MemCpy(pbyDest:=ADR(EncPosition[jointIdx]), 
					pbySrc:=ADR(pabyRxBuffer[bufferIdx]), 
					dwSize:=SIZEOF(EncPosition[jointIdx]));
	bufferIdx := bufferIdx + 4;
END_FOR

// index 25 will be for limit switch inputs
rx_j1_limit := pabyRxBuffer[25].0;
rx_j2_limit := pabyRxBuffer[25].1;
rx_j3_limit := pabyRxBuffer[25].2;
rx_j4_limit := pabyRxBuffer[25].3;
rx_j5_limit := pabyRxBuffer[25].4;
rx_j6_limit := pabyRxBuffer[25].5;
//rx_ := pabyRxBuffer[25].6;
//rx_ := pabyRxBuffer[25].7;

//rx_ := pabyRxBuffer[27];
//rx_ := pabyRxBuffer[28];
//rx_ := pabyRxBuffer[29];
//rx_ := pabyRxBuffer[30];
//rx_ := pabyRxBuffer[31];

// index 31 will be for gpio byte (bits 0 through 7)
GVL.DigitalInput[0] := pabyRxBuffer[31].0;
GVL.DigitalInput[1] := pabyRxBuffer[31].1;
GVL.DigitalInput[2] := pabyRxBuffer[31].2;
GVL.DigitalInput[3] := pabyRxBuffer[31].3;
GVL.DigitalInput[4] := pabyRxBuffer[31].4;
GVL.DigitalInput[5] := pabyRxBuffer[31].5;
GVL.DigitalInput[6] := pabyRxBuffer[31].6;
GVL.DigitalInput[7] := pabyRxBuffer[31].7;

M_HandleDriveIO();
                  

METHOD PUBLIC M_HandleDriveIO

VAR
END_VAR

VAR_INPUT
END_VAR

VAR_OUTPUT
END_VAR

VAR CONSTANT
END_VAR
                          (*                    DMT542T Stepper Driver
	Pulse and Direction Connection:
	(1) Optically isolated, high level 4.5-5V or 24V, low voltage 0-0.5V
	(2) Maximum 200 KHz input frequency
	(3) The width of PUL signal is at least 2.5μs, duty cycle is recommended 50%
	(4) DIR signal requires advance PUL signal minimum 5 μs in single pulse mode
	(5) The factory setting of control signal voltage is 24V, must need to set S2 (figure 2) if it is 5V
	
	Enable Connection: (default no connection)
	(1) Optically isolated, differential.
	(2) Disable the drive by 4.5- 24V input connection; enable the drive by 0-0.5V connection (3) ENA signal requires advance DIR signal minimum 5μs in single pulse mode
	(4) Enable time to be at least 200ms
*)
(*
	J1 - 400 steps per revolution
	J2 - 400 steps per revolution
	J3 - 400 steps per revolution
	J4 - 400 steps per revolution
	J5 - 800 steps per revolution
	J6 - 400 steps per revolution
*)

SM_Drive_PosControl_J1.in.dwActPosition := DINT_TO_DWORD(EncPosition[0]);
SM_Drive_PosControl_J2.in.dwActPosition := DINT_TO_DWORD(EncPosition[1]);
SM_Drive_PosControl_J3.in.dwActPosition := DINT_TO_DWORD(EncPosition[2]);
SM_Drive_PosControl_J4.in.dwActPosition := DINT_TO_DWORD(-EncPosition[3]);
SM_Drive_PosControl_J5.in.dwActPosition := DINT_TO_DWORD(EncPosition[4]);
SM_Drive_PosControl_J6.in.dwActPosition := DINT_TO_DWORD(EncPosition[5]);

SM_Drive_PosControl_J1.bHWLimitEnable := NOT _00_Main.SMC_Homing_J1.bBusy;
SM_Drive_PosControl_J2.bHWLimitEnable := NOT _00_Main.SMC_Homing_J2.bBusy;
SM_Drive_PosControl_J3.bHWLimitEnable := NOT _00_Main.SMC_Homing_J3.bBusy;
SM_Drive_PosControl_J4.bHWLimitEnable := NOT _00_Main.SMC_Homing_J4.bBusy;
SM_Drive_PosControl_J5.bHWLimitEnable := NOT _00_Main.SMC_Homing_J5.bBusy;
SM_Drive_PosControl_J6.bHWLimitEnable := NOT _00_Main.SMC_Homing_J6.bBusy;

SM_Drive_PosControl_J1.in.bLimitNeg := TRUE;
SM_Drive_PosControl_J2.in.bLimitNeg := TRUE;
SM_Drive_PosControl_J3.in.bLimitNeg := rx_j3_limit;
SM_Drive_PosControl_J4.in.bLimitNeg := rx_j4_limit;
SM_Drive_PosControl_J5.in.bLimitNeg := rx_j5_limit;
SM_Drive_PosControl_J6.in.bLimitNeg := TRUE;

SM_Drive_PosControl_J1.in.bLimitPos := rx_j1_limit;
SM_Drive_PosControl_J2.in.bLimitPos := rx_j2_limit;
SM_Drive_PosControl_J3.in.bLimitPos := TRUE;
SM_Drive_PosControl_J4.in.bLimitPos := TRUE;
SM_Drive_PosControl_J5.in.bLimitPos := TRUE;
SM_Drive_PosControl_J6.in.bLimitPos := rx_j6_limit;

SM_Drive_PosControl_J1.in.bDriveStartRealState := rx_en;
SM_Drive_PosControl_J1.in.bRegulatorRealState := rx_en;
SM_Drive_PosControl_J2.in.bDriveStartRealState := rx_en;
SM_Drive_PosControl_J2.in.bRegulatorRealState := rx_en;
SM_Drive_PosControl_J3.in.bDriveStartRealState := rx_en;
SM_Drive_PosControl_J3.in.bRegulatorRealState := rx_en;
SM_Drive_PosControl_J4.in.bDriveStartRealState := rx_en;
SM_Drive_PosControl_J4.in.bRegulatorRealState := rx_en;
SM_Drive_PosControl_J5.in.bDriveStartRealState := rx_en;
SM_Drive_PosControl_J5.in.bRegulatorRealState := rx_en;
SM_Drive_PosControl_J6.in.bDriveStartRealState := rx_en;
SM_Drive_PosControl_J6.in.bRegulatorRealState := rx_en;

// convert degrees per second to revolutions per second as that is what the drives take
SetVelocity[0] := LREAL_TO_REAL(-SM_Drive_PosControl_J1.out.fSetVelocity / 360.0); 
SetVelocity[1] := LREAL_TO_REAL(SM_Drive_PosControl_J2.out.fSetVelocity / 360.0);
SetVelocity[2] := LREAL_TO_REAL(SM_Drive_PosControl_J3.out.fSetVelocity / 360.0);
SetVelocity[3] := LREAL_TO_REAL(SM_Drive_PosControl_J4.out.fSetVelocity / 360.0);
SetVelocity[4] := LREAL_TO_REAL(SM_Drive_PosControl_J5.out.fSetVelocity / 360.0);
SetVelocity[5] := LREAL_TO_REAL(SM_Drive_PosControl_J6.out.fSetVelocity / 360.0);

tx_en := GVL.PowerOn;

                        
END_METHOD
END_PROGRAM

FUNCTION_BLOCK JogProcessor
VAR_IN_OUT
	AxisGroup: AXIS_GROUP_REF_SM3;
END_VAR

VAR_INPUT
	Enable: BOOL;
	Reset: BOOL;
END_VAR

VAR_OUTPUT
	ABC_as_ACS: BOOL;
	CoordSystem: SMC_COORD_SYSTEM;
	Position: SMC_POS_REF;
	Done: BOOL;
	Busy: BOOL;
	Error: BOOL;
	ErrorID: SMC_ERROR;
END_VAR

VAR
	_ExecuteRtrig: R_TRIG;
	_ExecuteFtrig: F_TRIG;
	_ResetRtrig: R_TRIG;
	_ErrorRtrig: R_TRIG;
	
	_SequenceMain: INT;
	
	_SMC_GroupJog2: SMC_GroupJog2;
	_SMC_GroupPower: SMC_GroupPower;
	_GroupPower: BOOL;
	_MC_GroupEnable: MC_GroupEnable;
	_MC_GroupDisable: MC_GroupDisable;
	_MC_GroupReset: MC_GroupReset;
	_MC_GroupReadActualPosition: MC_GroupReadActualPosition;
	_SMC_SetKinConfiguration: SMC_SetKinConfiguration;
	
	_FirstScan: BOOL:=TRUE;
	
END_VAR

VAR CONSTANT
	STEP_DONE: 				INT := 1000;
	STEP_IDLE: 				INT := 0000;
	STEP_GROUP_POWER_ON: 	INT := 0022;
	STEP_WAIT_POWER_ON: 	INT := 0024;
	STEP_GROUP_ENABLE: 		INT := 0030;
	STEP_WAIT_ENABLE: 		INT := 0035;
	STEP_READ_POSITION: 	INT := 0040;
	STEP_WAIT_POSITION: 	INT := 0050;
	STEP_SET_KINEMATICS: 	INT := 0060;
	STEP_WAIT_KINEMATICS: 	INT := 0070;
	STEP_JOG:				INT := 0080;
	STEP_WAIT_JOG:			INT := 0090;
	STEP_GROUP_DISABLE: 	INT := 0100;
	STEP_WAIT_DISABLE: 		INT := 0110;
	STEP_GROUP_POWER_OFF: 	INT := 0120;
END_VAR

                    _ExecuteRtrig(CLK:=_SMC_GroupJog2.Enable);
_ExecuteFtrig(CLK:=_SMC_GroupJog2.Enable);
_ResetRtrig(CLK:=Reset);

IF _FirstScan THEN
	_FirstScan := FALSE;
	_SMC_GroupJog2.Velocity := 10.0;
	_SMC_GroupJog2.Acceleration := 300.0;
	_SMC_GroupJog2.Deceleration := 300.0;
	_SMC_GroupJog2.Jerk := 1000.0;
	_SMC_GroupJog2.MaxAngularDistance := 90.0;
	_SMC_GroupJog2.MaxLinearDistance := 100.0;
	_SMC_GroupJog2.AccFactor := 1.0;
	_SMC_GroupJog2.VelFactor := 0.1;
	_SMC_GroupJog2.JerkFactor := 1.0;
	_SMC_GroupJog2.TorqueFactor := 1.0;
	_SMC_GroupJog2.CoordSystem := SMC_COORD_SYSTEM.MCS;
	
END_IF

CASE _SequenceMain OF
	STEP_DONE: // done
		_GroupPower := FALSE;
  		_MC_GroupEnable.Execute := FALSE;
  		_MC_GroupDisable.Execute := FALSE;
		_MC_GroupReset.Execute := FALSE;
  		_MC_GroupReadActualPosition.Enable := FALSE;
		_SMC_SetKinConfiguration.Execute := FALSE;
		Busy := FALSE;
		Done := TRUE;
		_SequenceMain := STEP_IDLE;
		
	STEP_IDLE: // IDLE
		IF _ExecuteRtrig.Q AND Enable THEN
			Busy := TRUE;
			Done := FALSE;
			_SequenceMain := STEP_GROUP_POWER_ON;
		END_IF
		
	STEP_GROUP_POWER_ON:
		_GroupPower := TRUE;
		_SequenceMain := STEP_WAIT_POWER_ON;
		
	STEP_WAIT_POWER_ON:
		IF _SMC_GroupPower.Error THEN
			Error := TRUE;
			ErrorID := _SMC_GroupPower.ErrorID;
		ELSIF _SMC_GroupPower.Status THEN
			_SequenceMain := STEP_GROUP_ENABLE;
		END_IF
		
	STEP_GROUP_ENABLE:
		_MC_GroupEnable.Execute := TRUE;
		_SequenceMain := STEP_WAIT_ENABLE;
		
	STEP_WAIT_ENABLE:
		IF NOT _MC_GroupEnable.Busy THEN // this is a hack. we need to figure out is the group is already enabled first
			_SequenceMain := STEP_READ_POSITION;
		END_IF;
		
	STEP_READ_POSITION: // read group position
		_MC_GroupReadActualPosition.Enable := TRUE;
		_SequenceMain := STEP_WAIT_POSITION;
		
	STEP_WAIT_POSITION: // wait for group read position
		IF _MC_GroupReadActualPosition.Error THEN
			Error := TRUE;
			ErrorID := _MC_GroupReadActualPosition.ErrorID;
		ELSIF _MC_GroupReadActualPosition.Valid THEN
			_SequenceMain := STEP_SET_KINEMATICS;
		END_IF
		
	STEP_SET_KINEMATICS: // set kinematics
		_SMC_SetKinConfiguration.Execute := TRUE;
		_SequenceMain := STEP_WAIT_KINEMATICS;
		
	STEP_WAIT_KINEMATICS: // wait for set kinematics
		IF _SMC_SetKinConfiguration.Error THEN
			Error := TRUE;
			ErrorID := _SMC_SetKinConfiguration.ErrorID;
		ELSIF _SMC_SetKinConfiguration.Done THEN
			_SMC_SetKinConfiguration.Execute := FALSE;
			_SequenceMain := STEP_JOG;
		END_IF
		
	STEP_JOG: //
		_SequenceMain := STEP_WAIT_JOG;
		
	STEP_WAIT_JOG: //
		IF _SMC_GroupJog2.Error THEN
			Error := TRUE;
			ErrorID := _SMC_GroupJog2.ErrorID;
		END_IF
		IF _ExecuteFtrig.Q THEN
			_SequenceMain := STEP_GROUP_DISABLE;
		END_IF
		
	STEP_GROUP_DISABLE:
		_MC_GroupDisable.Execute := TRUE;
		_SequenceMain := STEP_WAIT_DISABLE;
		
	STEP_WAIT_DISABLE:
		IF NOT _MC_GroupDisable.Busy THEN // this is a hack. we need to figure out is the group is already disabled first
			_SequenceMain := STEP_GROUP_POWER_OFF;
		END_IF
		
	STEP_GROUP_POWER_OFF:
		_GroupPower := FALSE;
		_SequenceMain := STEP_DONE;
	
END_CASE

IF _ResetRtrig.Q AND Error THEN
	Error := FALSE;
	ErrorID := SMC_NO_ERROR;
	_MC_GroupReset.Execute := TRUE;
	_MC_GroupDisable.Execute := TRUE;
	_SequenceMain := STEP_DONE;
END_IF

_SMC_GroupPower(
	AxisGroup:= AxisGroup, 
	Enable:= _GroupPower, 
	bRegulatorOn:= _GroupPower, 
	bDriveStart:= _GroupPower, 
	Status=> , 
	Busy=> , 
	Error=> , 
	ErrorID=> );

_MC_GroupEnable(
	AxisGroup:= AxisGroup, 
	Execute:= , 
	CompatibilityOptions:= , 
	Done=> , 
	Busy=> , 
	Error=> , 
	ErrorID=> );
	
_MC_GroupDisable(
	AxisGroup:= AxisGroup, 
	Execute:= , 
	Done=> , 
	Busy=> , 
	Error=> , 
	ErrorID=> );

_MC_GroupReset(
	AxisGroup:= AxisGroup, 
	Execute:= , 
	Done=> , 
	Busy=> , 
	Error=> , 
	ErrorID=> );

_MC_GroupReadActualPosition(
	AxisGroup:= AxisGroup, 
	Enable:= , 
	CoordSystem:= _SMC_GroupJog2.CoordSystem, 
	Valid=> , 
	Busy=> , 
	Error=> , 
	ErrorID=> , 
	Position=> , 
	KinematicConfig=> );
	
_SMC_SetKinConfiguration(
	AxisGroup:= AxisGroup, 
	Execute:= , 
	ConfigData:= _MC_GroupReadActualPosition.KinematicConfig, 
	Done=> , 
	Busy=> , 
	Error=> , 
	ErrorID=> );

_SMC_GroupJog2(
	AxisGroup:= AxisGroup, 
	Enable:= , 
	Forward:= , 
	Backward:= , 
	MaxLinearDistance:= , 
	MaxAngularDistance:= , 
	Velocity:= , 
	Acceleration:= , 
	Deceleration:= , 
	Jerk:= , 
	VelFactor:= , //_SMC_GroupJog2.Velocity / 100.0, 
	AccFactor:= , 
	JerkFactor:= , 
	TorqueFactor:= , 
	CoordSystem:= , 
	ABC_as_ACS:= , 
	Active=> , 
	Busy=> , 
	Error=> , 
	ErrorID=> , 
	CurrentPosition=> Position);
	CoordSystem := _SMC_GroupJog2.CoordSystem;
	ABC_as_ACS := _SMC_GroupJog2.ABC_as_ACS;
	
_ErrorRtrig(CLK:=_SMC_GroupPower.Error
				OR _MC_GroupReadActualPosition.Error
				OR _SMC_SetKinConfiguration.Error
				OR _SMC_GroupJog2.Error);
				
IF _ErrorRtrig.Q THEN
	Error := TRUE;
END_IF

                  
END_FUNCTION_BLOCK

FUNCTION_BLOCK CommandProcessor EXTENDS Module
VAR_IN_OUT
	AxisGroup: AXIS_GROUP_REF_SM3;
	Servo1: AXIS_REF_SM3;
	Servo2: AXIS_REF_SM3;
END_VAR
VAR_INPUT
	Enable: BOOL;
	Commands: ARRAY [GVL.PROG_CMDS_ARR_BEG..GVL.PROG_CMDS_ARR_END] OF DUT_Command;
END_VAR
VAR_OUTPUT
	ItfActiveProcessorUnitMode	: PACK_ML.IUnitMode;
	ItfActiveModule: ItfModule;
	ActiveCommand: DUT_Command;
	StatusText: STRING(255);
END_VAR
VAR
	_Commands: ARRAY [GVL.PROG_CMDS_ARR_BEG..GVL.PROG_CMDS_ARR_END] OF DUT_Command;
	_DummyUnitMode: PACK_ML.UnitMode;
	_UnitModeCurrentState: PACK_ML.State;
	//_SequenceMain, _SeqAborting, _SeqClearing, _SeqResetting: INT;
	_CurrentCmdIdx: UINT;
	_ProcessMoveCommand: MoveCmdProcessor;
	_ProcessPauseCommand: PauseCmdProcessor;
	//_ProcessInputCommand: InputCommandProcessor;
	_ProcessOutputCommand: OutputCmdProcessor;
	_ProcessorDoneRtrig: R_TRIG;
    _ProcessVisionCommand: REFERENCE TO VisionCmdProcessor; // keep vision in separate task
	_ProcessVarSetCommand: VarSetCmdProcessor;
	_ProcessCncCommand: CncCmdProcessor;
	_ProcessLogicCommand: LogicCmdProcessor;
	_FirstScan: BOOL:=TRUE;
END_VAR

VAR CONSTANT
	_STEP_DONE: 			INT := 1000;
	_STEP_IDLE: 			INT := 0000;
	_STEP_CMD:				INT := 0010;
	_STEP_WAIT:				INT := 0020;
	_STEP_ERR:              INT := 0030;
END_VAR

                    // keep this reference at the top in case we reference this somewhere else first
// hint: originally this was an issue because of the done and reset bits being referenced first
_ProcessVisionCommand REF= _40_Vision.ProcessVisionCommand;

//
SUPER^();

//
IF _FirstScan THEN
	// will exception if we don't set this on first scan
	_DummyUnitMode(sName := 'Active Processor', 
					eInitialState := PACK_ML.State.Idle,
					xActive := TRUE);
	ItfActiveProcessorUnitMode := _DummyUnitMode;
END_IF

// this is at best a hack and needs to be rethought out.
// we logically cant assign a process as the active unit mode 
// at start up so we use this dummy one
CASE _DummyUnitMode.CurrentState OF
	PACK_ML.State.Stopped,
	PACK_ML.State.Aborted,
	PACK_ML.State.Held,
	PACK_ML.State.Suspended,
	PACK_ML.State.Complete,
	PACK_ML.State.Idle:
		//
	PACK_ML.State.Resetting,
	PACK_ML.State.Starting,
	PACK_ML.State.Execute,
	PACK_ML.State.Suspending,
	PACK_ML.State.UnSuspending,
	PACK_ML.State.Holding,
	PACK_ML.State.UnHolding,
	PACK_ML.State.Completing,
	PACK_ML.State.Aborting,
	PACK_ML.State.Stopping,
	PACK_ML.State.Clearing:
		_DummyUnitMode.ActingStateCompleted();
END_CASE

// PackML state machine implementation
_UnitModeCurrentState := SUPER^._UnitMode.CurrentState;

//
IF _ProcessMoveCommand.Error THEN
	SUPER^.M_Error(Description:=CONCAT('Move Error: ', _ProcessMoveCommand.ErrorDescription));
	StatusText:=SUPER^.ErrorDescription;
END_IF
IF _ProcessPauseCommand.Error THEN
	SUPER^.M_Error(Description:=CONCAT('Pause Error: ', _ProcessPauseCommand.ErrorDescription));
	StatusText:=SUPER^.ErrorDescription;
END_IF
(*IF _ProcessInputCommand.Error THEN
	SUPER^._M_Error(Description:=CONCAT('Input Error: ', _ProcessInputCommand.ErrorDescription));
	StatusText:=SUPER^.ErrorDescription;
END_IF*)
IF _ProcessOutputCommand.Error THEN
	SUPER^.M_Error(Description:=CONCAT('Output Error: ', _ProcessOutputCommand.ErrorDescription));
	StatusText:=SUPER^.ErrorDescription;
END_IF       
IF _ProcessVisionCommand.Error THEN
	SUPER^.M_Error(Description:=CONCAT('Vision Error: ', _ProcessVisionCommand.ErrorDescription));
	StatusText:=SUPER^.ErrorDescription;
END_IF
IF _ProcessVarSetCommand.Error THEN
	SUPER^.M_Error(Description:=CONCAT('Variable Error: ', _ProcessVarSetCommand.ErrorDescription));
	StatusText:=SUPER^.ErrorDescription;
END_IF
IF _ProcessCncCommand.Error THEN
	SUPER^.M_Error(Description:=CONCAT('CNC Error: ', _ProcessCncCommand.ErrorDescription));
	StatusText:=SUPER^.ErrorDescription;
END_IF
IF _ProcessLogicCommand.Error THEN
	SUPER^.M_Error(Description:=CONCAT('Logic Error: ', _ProcessLogicCommand.ErrorDescription));
	StatusText:=SUPER^.ErrorDescription;
END_IF

_ProcessMoveCommand(
	StoredPositions:= SUPER^.StoredPositions,
	VisionRegisters:= SUPER^.VisionRegisters,
	Flags:= SUPER^.Flags,
	AxisGroup:= AxisGroup, 
	Acceleration:= 1000, 
	AccFactor:= 0.05,
	Jerk:= 1000,
	JerkFactor:= 1, 
	Position=> ,
	ItfUnitMode=>, 
	Error=> );

_ProcessPauseCommand(
	StoredPositions:= SUPER^.StoredPositions,
	VisionRegisters:= SUPER^.VisionRegisters,
	Flags:= SUPER^.Flags, 
	ElapsedTime=> , 
	RemainingTime=> , 
	ItfUnitMode=>, 
	Error=> );

//_ProcessInputCommand();
_ProcessOutputCommand(
	StoredPositions:= SUPER^.StoredPositions,
	VisionRegisters:= SUPER^.VisionRegisters,
	Flags:= SUPER^.Flags,
	Outputs:= GVL.DigitalOutput,
	Servo1:= Servo1, 
	Servo2:= Servo2, 
	Enable:= Enable,
	ItfUnitMode=>, 
	Error=> );
	
_ProcessVarSetCommand( 
	StoredPositions:= SUPER^.StoredPositions,
	VisionRegisters:= SUPER^.VisionRegisters,
	Flags:= SUPER^.Flags,
	ItfUnitMode=>, 
	Error=> , 
	ErrorDescription=> );

_ProcessCncCommand(
	StoredPositions:= SUPER^.StoredPositions,
	VisionRegisters:= SUPER^.VisionRegisters,
	Flags:= SUPER^.Flags,
	AxisGroup:= AxisGroup, 
	SM3_Drive_PosControl_J1:=SM_Drive_PosControl_J1,
	SM3_Drive_PosControl_J2:=SM_Drive_PosControl_J2,
	SM3_Drive_PosControl_J3:=SM_Drive_PosControl_J3,
	SM3_Drive_PosControl_J4:=SM_Drive_PosControl_J4,
	SM3_Drive_PosControl_J5:=SM_Drive_PosControl_J5,
	SM3_Drive_PosControl_J6:=SM_Drive_PosControl_J6,
	GapVelocity:= , 
	AvoidGaps:= , 
	GapAccel:= , 
	ItfUnitMode=>, 
	Error=> , 
	ErrorDescription=> );
	
_ProcessLogicCommand(
	StoredPositions:= SUPER^.StoredPositions,
	VisionRegisters:= SUPER^.VisionRegisters,
	Flags:= SUPER^.Flags,
	CmdProcessor:= THIS^,
	ItfUnitMode=>, 
	Error=> , 
	ErrorDescription=> , 
	CmdIO:= GVL.CmdIO);
	
	_FirstScan := FALSE;
                  

METHOD PROTECTED M_Complete : BOOL
                          // once complete, reset to get back to idle
SUPER^._UnitMode.Reset();
                        
END_METHOD

METHOD PROTECTED M_Resetting : BOOL
                          CASE _SeqResetting OF
	0:
		_ProcessMoveCommand.M_Home();
		_ProcessPauseCommand.M_Home();
		//_ProcessInputCommand.M_Home();
		_ProcessOutputCommand.M_Home();
		_ProcessVisionCommand.M_Home();
		_ProcessVarSetCommand.M_Home();
		_ProcessCncCommand.M_Home();
		_ProcessLogicCommand.M_Home();
		_SeqResetting := _SeqResetting + 1;
	1:
		IF _ProcessMoveCommand.PropCurrentState = PACK_ML.State.Idle
			AND _ProcessPauseCommand.PropCurrentState = PACK_ML.State.Idle 
			//AND _ProcessInputCommand.PropCurrentState = PACK_ML.State.Idle
			AND _ProcessOutputCommand.PropCurrentState = PACK_ML.State.Idle
			AND _ProcessVisionCommand.PropCurrentState = PACK_ML.State.Idle
			AND _ProcessVarSetCommand.PropCurrentState = PACK_ML.State.Idle
			AND _ProcessCncCommand.PropCurrentState = PACK_ML.State.Idle
			AND _ProcessLogicCommand.PropCurrentState = PACK_ML.State.Idle THEN
				_SeqResetting := 0;
				SUPER^.M_StateComplete();
		END_IF
		
END_CASE

SUPER^.M_Reset();

(*IF ItfActiveModule <> 0 THEN
	CASE _Seq OF
		0:
			IF NOT ItfActiveModule.PropCurrentState = PACK_ML.State.Idle THEN
				ItfActiveModule.M_Home();
				_Seq := 1;
			ELSE
				SUPER^.M_StateComplete();
			END_IF
		1:
			IF ItfActiveModule.PropCurrentState = PACK_ML.State.Idle THEN
				_Seq := 0;
			END_IF
			
	END_CASE
	
ELSE
	SUPER^.M_StateComplete();
	_Seq := 0;
	
END_IF*)
                        
END_METHOD

METHOD PUBLIC M_SetNextCommand : BOOL // returns true if successful
VAR_INPUT
	CommandNumber: UINT;
END_VAR
                          IF CommandNumber <= GVL.PROG_CMDS_ARR_END AND CommandNumber >= GVL.PROG_CMDS_ARR_BEG THEN
	_CurrentCmdIdx := CommandNumber;
	M_SetNextCommand := TRUE;
ELSE
	M_SetNextCommand := FALSE;
END_IF
                        
END_METHOD

METHOD PROTECTED M_Idle : BOOL
                          // in this state, we want to reset all the function blocks and hang out
_SeqMain := _STEP_IDLE;
_SeqAborting := 0;
_SeqClearing := 0;
_SeqResetting := 0;
                        
END_METHOD

METHOD PROTECTED M_SetPackML : BOOL
                          // SUPER already does this but the default is eInitialState:=PACK_ML.State.Idle 
// and we want PACK_ML.State.Aborted for the Orchestrator
SUPER^._UnitMode(sName := 'Orchestrator',
				eInitialState := PACK_ML.State.Aborted,
				xActive := TRUE);
                        
END_METHOD

METHOD PROTECTED M_Starting : BOOL
                          // here we want to clear things and get ready for the execute state
// we can consider this the "INIT" state
_CurrentCmdIdx := 0;
_SeqMain := _STEP_CMD;
_Commands := Commands;
SUPER^.M_StateComplete();
                        
END_METHOD

METHOD PROTECTED M_Execute : BOOL
                          // here we want to execute our commands/jobs/etc and set completed when done.
//
CASE _SeqMain OF
  	_STEP_DONE:
		_SeqMain := _STEP_IDLE;
		
	_STEP_IDLE:
		// hang out here until called to run
		_CurrentCmdIdx := 0;
		SUPER^.M_StateComplete();
		
	_STEP_CMD: //
		IF _CurrentCmdIdx <= GVL.PROG_CMDS_ARR_END AND _CurrentCmdIdx >= GVL.PROG_CMDS_ARR_BEG THEN
			//
			IF Commands[_CurrentCmdIdx].CommandType = DUT_CommandType.Disabled THEN
				// want to increment here so that we can disable some commands 
				// in the program and it continue to execute
				_CurrentCmdIdx := _CurrentCmdIdx + 1;
				_SeqMain := _STEP_CMD;
				
			ELSE
				CASE Commands[_CurrentCmdIdx].CommandType OF
					DUT_CommandType.MoveCommand: //
						StatusText := 'Move Command in Progress.';
						ItfActiveProcessorUnitMode := _ProcessMoveCommand.ItfUnitMode;
						ItfActiveModule := _ProcessMoveCommand;
						_ProcessMoveCommand.Command := Commands[_CurrentCmdIdx].CommandString;
						ItfActiveModule.M_Start();
					
					DUT_CommandType.PauseCommand: //
						StatusText := 'Pause Command in Progress.';
						ItfActiveProcessorUnitMode := _ProcessPauseCommand.ItfUnitMode;
						ItfActiveModule := _ProcessPauseCommand;
						_ProcessPauseCommand.Command := Commands[_CurrentCmdIdx].CommandString;
						ItfActiveModule.M_Start();
					
					DUT_CommandType.InputCommand: //
						StatusText := 'Input Command in Progress.';
						//ActiveUnitMode := _ProcessInputCommand.ItfUnitMode;
						//ItfActiveModule := _ProcessInputCommand;
						//_ProcessInputCommand.Command := Commands[_CurrentCmdIdx].CommandString;
						//ItfActiveModule.M_Start();
					
					DUT_CommandType.OutputCommand: //
						StatusText := 'Output Command in Progress.';
						ItfActiveProcessorUnitMode := _ProcessOutputCommand.ItfUnitMode;
						ItfActiveModule := _ProcessOutputCommand;
						_ProcessOutputCommand.Command := Commands[_CurrentCmdIdx].CommandString;
						ItfActiveModule.M_Start();
					
					DUT_CommandType.VisionCommand: //
						StatusText := 'Vision Command in Progress.';
						ItfActiveProcessorUnitMode := _ProcessVisionCommand.ItfUnitMode;
						ItfActiveModule := _ProcessVisionCommand;
						_ProcessVisionCommand.Command := Commands[_CurrentCmdIdx].CommandString;
						ItfActiveModule.M_Start();
					
					DUT_CommandType.VarSetCommand: //
						StatusText := 'VarSet Command in Progress.';
						ItfActiveProcessorUnitMode := _ProcessVarsetCommand.ItfUnitMode;
						ItfActiveModule := _ProcessVarsetCommand;
						_ProcessVarsetCommand.Command := Commands[_CurrentCmdIdx].CommandString;
						ItfActiveModule.M_Start();
					
					DUT_CommandType.CncCommand: //
						StatusText := 'CNC Command in Progress.';
						ItfActiveProcessorUnitMode := _ProcessCncCommand.ItfUnitMode;
						ItfActiveModule := _ProcessCncCommand;
						_ProcessCncCommand.Command := Commands[_CurrentCmdIdx].CommandString;
						ItfActiveModule.M_Start();
					
					DUT_CommandType.LogicCommand: //
						StatusText := 'Logic Command in Progress.';
						ItfActiveProcessorUnitMode := _ProcessLogicCommand.ItfUnitMode;
						ItfActiveModule := _ProcessLogicCommand;
						_ProcessLogicCommand.Command := Commands[_CurrentCmdIdx].CommandString;
						ItfActiveModule.M_Start();
						
				ELSE
					_SeqMain := _STEP_CMD;
					
				END_CASE
				
				// wait for executing
				IF ItfActiveModule.PropCurrentState = PACK_ML.State.Execute THEN
					ActiveCommand := Commands[_CurrentCmdIdx];
					_CurrentCmdIdx := _CurrentCmdIdx + 1;
					_SeqMain := _STEP_WAIT;
				END_IF
			END_IF
				
		ELSE
			_SeqMain := _STEP_DONE;
		END_IF
		
	_STEP_WAIT: // wait for command to finish
		//
		IF _ProcessorDoneRtrig.Q THEN
			_SeqMain := _STEP_CMD;
		END_IF
		//
		IF ItfActiveModule.PropError THEN
			SUPER^._UnitMode.Suspend();
			_SeqMain := _STEP_ERR;
		END_IF
		
	_STEP_ERR: //
	
END_CASE

// watch for rising edge of idle state. this was done for all processors since 
// the vision processor runs in a separate task and isnt guaranteed to start in the same 
// PLC scan.
_ProcessorDoneRtrig(clk:=ItfActiveProcessorUnitMode.CurrentState = PACK_ML.State.Idle);
                        
END_METHOD

METHOD PROTECTED M_Suspending : BOOL
                          IF ItfActiveModule <> 0 THEN
	IF ItfActiveModule.PropCurrentState = PACK_ML.State.Execute THEN
		ItfActiveModule.M_Hold();
		IF ItfActiveModule.PropCurrentState = PACK_ML.State.Held THEN
			SUPER^.M_StateComplete();
		END_IF
	ELSE
		SUPER^.M_StateComplete();
	END_IF
	
ELSE
	SUPER^.M_StateComplete();
	
END_IF
                        
END_METHOD

METHOD PROTECTED M_UnSuspending : BOOL
                          //
IF ItfActiveModule <> 0 THEN
	ItfActiveModule.M_Start();
	IF ItfActiveModule.PropCurrentState = PACK_ML.State.Execute THEN
		SUPER^.M_StateComplete();
	END_IF
	
ELSE
	SUPER^.M_StateComplete();
	
END_IF

//
_SeqMain := _STEP_WAIT;
                        
END_METHOD

METHOD PROTECTED M_Holding : BOOL
                          IF ItfActiveModule <> 0 THEN
	ItfActiveModule.M_Hold();
	IF ItfActiveModule.PropCurrentState = PACK_ML.State.Held THEN
		SUPER^.M_StateComplete();
	END_IF
ELSE
	SUPER^.M_StateComplete();
END_IF
                        
END_METHOD

METHOD PROTECTED M_Unholding : BOOL
                          //
IF ItfActiveModule <> 0 THEN
	ItfActiveModule.M_Start();
	IF ItfActiveModule.PropCurrentState = PACK_ML.State.Execute THEN
		SUPER^.M_StateComplete();
	END_IF
	
ELSE
	SUPER^.M_StateComplete();
	
END_IF

//
_SeqMain := _STEP_WAIT;
                        
END_METHOD

METHOD PROTECTED M_Aborting : BOOL
                          CASE _SeqAborting OF
	0:
		_ProcessMoveCommand.M_Abort();
		_ProcessPauseCommand.M_Abort();
		//_ProcessInputCommand.M_Abort();
		_ProcessOutputCommand.M_Abort();
		_ProcessVisionCommand.M_Abort();
		_ProcessVarSetCommand.M_Abort();
		_ProcessCncCommand.M_Abort();
		_ProcessLogicCommand.M_Abort();
		_SeqAborting := _SeqAborting + 1;
	1:
		IF _ProcessMoveCommand.PropCurrentState = PACK_ML.State.Aborted
			AND _ProcessPauseCommand.PropCurrentState = PACK_ML.State.Aborted 
			//AND _ProcessInputCommand.PropCurrentState = PACK_ML.State.Aborted
			AND _ProcessOutputCommand.PropCurrentState = PACK_ML.State.Aborted
			AND _ProcessVisionCommand.PropCurrentState = PACK_ML.State.Aborted
			AND _ProcessVarSetCommand.PropCurrentState = PACK_ML.State.Aborted
			AND _ProcessCncCommand.PropCurrentState = PACK_ML.State.Aborted
			AND _ProcessLogicCommand.PropCurrentState = PACK_ML.State.Aborted THEN
				_SeqAborting := 0;
				SUPER^.M_StateComplete();
		END_IF
		
END_CASE

(*IF ItfActiveModule <> 0 THEN
	ItfActiveModule.M_Abort();
	IF ItfActiveModule.PropCurrentState = PACK_ML.State.Aborted THEN
		SUPER^.M_StateComplete();
	END_IF
ELSE
	SUPER^.M_StateComplete();
END_IF*)
                        
END_METHOD

METHOD PROTECTED M_Stopping : BOOL
                          IF ItfActiveModule <> 0 THEN
	ItfActiveModule.M_Stop();
	IF ItfActiveModule.PropCurrentState = PACK_ML.State.Idle 
		OR ItfActiveModule.PropCurrentState = PACK_ML.State.Stopped 
		OR ItfActiveModule.PropCurrentState = PACK_ML.State.Aborted 
		OR ItfActiveModule.PropCurrentState = PACK_ML.State.Complete THEN
			SUPER^.M_StateComplete();
	END_IF
	
ELSE
	SUPER^.M_StateComplete();
	
END_IF
                        
END_METHOD

METHOD PROTECTED M_Clearing : BOOL
                          SUPER^.M_StateComplete();

(*IF SUPER^.Flags[GVL.HOME_COMPLETE].Value THEN
	CASE _SeqClearing OF
		0:
			_ProcessMoveCommand.M_Home();
			_SeqClearing := _SeqClearing + 1;
		1:
			IF _ProcessMoveCommand.PropCurrentState = PACK_ML.State.Idle THEN
				_SeqClearing := _SeqClearing + 1;
			END_IF
		2:
			IF NOT _ProcessMoveCommand.Error THEN
				_ProcessMoveCommand.Command := GVL.Pose2;
				_ProcessMoveCommand.M_Start();
				_SeqClearing := _SeqClearing + 1;
			ELSE
				SUPER^._M_Error(Description:='Move processor errored. Please reset and try again');
				_SeqClearing := -1;
			END_IF
		3:
			IF _ProcessMoveCommand.PropCurrentState = PACK_ML.State.Execute THEN
				_SeqClearing := _SeqClearing + 1;
			END_IF
		4:
			IF _ProcessMoveCommand.PropCurrentState = PACK_ML.State.Complete 
				OR _ProcessMoveCommand.PropCurrentState = PACK_ML.State.Stopped 
				OR _ProcessMoveCommand.PropCurrentState = PACK_ML.State.Aborted
				OR _ProcessMoveCommand.PropCurrentState = PACK_ML.State.Idle  THEN
					SUPER^.M_StateComplete();
					_SeqClearing := 0;
			END_IF
	END_CASE
ELSE
	SUPER^._M_Error(Description:='Drives are not homed. Please home and try again');
	_SeqClearing := -1;
END_IF

IF _ProcessMoveCommand.Error THEN
	SUPER^._M_Error(Description:='Move processor in error state. Please reset and try again');
	_SeqClearing := -1;
END_IF
*)

(*
IF ItfActiveModule <> 0 THEN
	//
	CASE _Seq OF
		0:
			IF NOT ItfActiveModule.PropCurrentState = PACK_ML.State.Stopped THEN
				ItfActiveModule.M_Abort();
				_Seq := 1;
			ELSE
				SUPER^.M_StateComplete();
			END_IF
		1:
			CASE ItfActiveModule.PropCurrentState OF
				PACK_ML.State.Aborted:
					ItfActiveModule.Clear();
				PACK_ML.State.Stopped:
					_Seq := 0;
			END_CASE
			
	END_CASE
ELSE
	_Seq := 0;
	SUPER^.M_StateComplete();
END_IF
*)

                        
END_METHOD
END_FUNCTION_BLOCK

FUNCTION_BLOCK ParseMoveCmd
VAR_INPUT
	Command: STRING(GVL.COMMAND_LEN);
END_VAR
VAR_OUTPUT
	stCommand: ST_MoveCmd;
	Error: BOOL:= FALSE;
	ErrorDescription: STRING:='';
END_VAR
VAR
	_CmdParams: ARRAY [0..GVL.COMMAND_LEN] OF STRING;
END_VAR
VAR CONSTANT
	_MoveTypeD: STRING(3):='DIR';
	_MoveTypeL: STRING(3):='LIN';
	_MoveTypeC: STRING(3):='CIR';
	_ChangeTypeA: STRING(3):='ABS';
	_ChangeTypeR: STRING(3):='REL';
	_CoordSystemAcs: STRING(3):='ACS';
	_CoordSystemMcs: STRING(3):='MCS';
	_CoordSystemPc1: STRING(3):='PC1';
	_CoordSystemPc2: STRING(3):='PC2';
	_CoordSystemTcs: STRING(3):='TCS';
	_CoordSystemWcs: STRING(3):='WCS';
	_CoordSystemIcs: STRING(3):='ICS';
	_CoordTypeH: STRING(3):='LIT';
	_CoordTypeV: STRING(3):='VAR';
	_ArrayTypeS: STRING(3):='STO';
	_ArrayTypeV: STRING(3):='VIS';
	_ArrayTypeF: STRING(3):='FLG';
	_CircleModeBor: STRING(3):='BOR';
	_CircleModeCen: STRING(3):='CEN';
	_CircleModeRad: STRING(3):='RAD';
	_PathChoiceClw: STRING(3):='CLW';
	_PathChoiceCcw: STRING(3):='CCW';
END_VAR

                    // D is direct move. L is linear move. C is a circular move
// R is relative position. A is absolute position
// V is variable coordinated. H is a hardcoded coordinated
// S is stored position array. V is vision register array.
// D|L|C R|A Speed CoordSystem X0000.00 Y0000.00 Z0000.00 A0000.00 B0000.00 C0000.00 BOR|CEN|RAD CCW|CLW X0000.00 Y0000.00 Z0000.00 A0000.00 B0000.00 C0000.00
// 'D A 10 MCS H +0250.00 +0000.00 +0500.00 +0000.00 +0045.00 +0180.00'
// 'C R 10 MCS H +0250.00 +0000.00 +0500.00 +0000.00 +0045.00 +0180.00 BOR CLW H +0250.00 +0000.00 +0500.00 +0000.00 +0045.00 +0180.00'
// 'D A 10 MCS V S 25'
// 'D A 10 MCS V V 33'
// 'C R 10 MCS V S 2 BOR CLW V S 005'
// 'C R 10 MCS V S 003 BOR CLW V V 006'
// 'C R 10 MCS V S 015 BOR CLW H +0250.00 +0000.00 +0500.00 +0000.00 +0045.00 +0180.00'
// 'C R 10 MCS H 250.0 0.0 500.0 0.0 45.0 180.0 BOR CLW V V 22'

Error := FALSE;
ErrorDescription := '';

// split command string into commands
_CmdParams:=F_SplitCmd(Command:=Command);

//
IF _CmdParams[0] = _MoveTypeD THEN
	stCommand.MoveType := DUT_Command_MoveType.DirectMove;
ELSIF _CmdParams[0] = _MoveTypeL THEN
	stCommand.MoveType := DUT_Command_MoveType.LinearMove;
ELSIF _CmdParams[0] = _MoveTypeC THEN
	stCommand.MoveType := DUT_Command_MoveType.CircularMove;
ELSE
	Error := TRUE;
	ErrorDescription := 'Incorrect move type';
END_IF

//
IF _CmdParams[1] = _ChangeTypeR THEN
	stCommand.PositionType := DUT_Command_PositionType.RelativePosition;
ELSIF _CmdParams[1] = _ChangeTypeA THEN
	stCommand.PositionType := DUT_Command_PositionType.AbsolutePosition;
ELSE
	Error := TRUE;
	ErrorDescription := 'Incorrect position type';
END_IF

//
stCommand.Speed := STRING_TO_LREAL(_CmdParams[2]);

//
IF _CmdParams[3] = _CoordSystemAcs THEN
	stCommand.CoordSystem := SMC_COORD_SYSTEM.ACS;
ELSIF _CmdParams[3] = _CoordSystemMcs THEN
	stCommand.CoordSystem := SMC_COORD_SYSTEM.MCS;
ELSIF _CmdParams[3] = _CoordSystemPc1 THEN
	stCommand.CoordSystem := SMC_COORD_SYSTEM.PCS_1;
ELSIF _CmdParams[3] = _CoordSystemPc2 THEN
	stCommand.CoordSystem := SMC_COORD_SYSTEM.PCS_2;
ELSIF _CmdParams[3] = _CoordSystemTcs THEN
	stCommand.CoordSystem := SMC_COORD_SYSTEM.TCS;
ELSIF _CmdParams[3] = _CoordSystemWcs THEN
	stCommand.CoordSystem := SMC_COORD_SYSTEM.WCS;
ELSIF _CmdParams[3] = _CoordSystemIcs THEN
	stCommand.CoordSystem := SMC_COORD_SYSTEM.ICS;
ELSE
	Error := TRUE;
	ErrorDescription := 'Incorrect coordinate system type';
END_IF

//
IF _CmdParams[4] = _CoordTypeH THEN
	stCommand.CoordinateType := DUT_Command_CoordinateType.Literal;
ELSIF _CmdParams[4] = _CoordTypeV THEN
	stCommand.CoordinateType := DUT_Command_CoordinateType.Variable;
ELSE
	Error := TRUE;
	ErrorDescription := 'Incorrect coordinate type'; // TODO wow i need a better name for this... wtf was i thinking?
END_IF

//
CASE stCommand.CoordinateType OF 
// 'D A 010 MCS H +0250.00 +0000.00 +0500.00 +0000.00 +0045.00 +0180.00'
	DUT_Command_CoordinateType.Literal:
		stCommand.CoordRef.X := STRING_TO_LREAL(_CmdParams[5]);
		stCommand.CoordRef.Y := STRING_TO_LREAL(_CmdParams[6]);
		stCommand.CoordRef.Z := STRING_TO_LREAL(_CmdParams[7]);
		stCommand.CoordRef.A := STRING_TO_LREAL(_CmdParams[8]);
		stCommand.CoordRef.B := STRING_TO_LREAL(_CmdParams[9]);
		stCommand.CoordRef.C := STRING_TO_LREAL(_CmdParams[10]);
// 'D A 010 MCS V S 001'
	DUT_Command_CoordinateType.Variable:
		stCommand.ArrayIndex := STRING_TO_UINT(_CmdParams[6]);
		IF stCommand.ArrayIndex <= GVL.POS_ARR_END 
			AND stCommand.ArrayIndex >= GVL.POS_ARR_BEG THEN
				IF _CmdParams[5] = _ArrayTypeS THEN
					stCommand.ArrayType := DUT_Command_ArrayType.StoredPosition;
					stCommand.CoordRef := PersistentVars.StoredPositions[stCommand.ArrayIndex].Position;
				ELSIF _CmdParams[5] = _ArrayTypeV THEN
					stCommand.ArrayType := DUT_Command_ArrayType.VisionRegister;
					stCommand.CoordRef := PersistentVars.VisionRegisters[stCommand.ArrayIndex].Position;
				ELSE
					Error := TRUE;
					ErrorDescription := 'Incorrect array type';
				END_IF
		ELSE
			Error := TRUE;
			ErrorDescription := 'Array index out of bounds';
		END_IF
	
END_CASE

//
CASE stCommand.CoordinateType OF 
// 'C R 010 MCS H +0250.00 +0000.00 +0500.00 +0000.00 +0045.00 +0180.00 BOR CLW H +0250.00 +0000.00 +0500.00 +0000.00 +0045.00 +0180.00'
	DUT_Command_CoordinateType.Literal:
		IF _CmdParams[11] = _CircleModeBor THEN
			stCommand.CircleMode := SMC_CIRC_MODE.BORDER;
		ELSIF _CmdParams[11] = _CircleModeCen THEN
			stCommand.CircleMode := SMC_CIRC_MODE.CENTER;
		ELSIF _CmdParams[11] = _CircleModeRad THEN
			stCommand.CircleMode := SMC_CIRC_MODE.RADIUS;
		ELSE
			Error := TRUE;
			ErrorDescription := 'Incorrect circle mode';
		END_IF
// 'C R 010 MCS V S 001 BOR CLW H +0250.00 +0000.00 +0500.00 +0000.00 +0045.00 +0180.00'
	DUT_Command_CoordinateType.Variable:
		IF _CmdParams[7] = _CircleModeBor THEN
			stCommand.CircleMode := SMC_CIRC_MODE.BORDER;
		ELSIF _CmdParams[7] = _CircleModeCen THEN
			stCommand.CircleMode := SMC_CIRC_MODE.CENTER;
		ELSIF _CmdParams[7] = _CircleModeRad THEN
			stCommand.CircleMode := SMC_CIRC_MODE.RADIUS;
		ELSE
			Error := TRUE;
			ErrorDescription := 'Incorrect circle mode';
		END_IF
	
END_CASE

//
CASE stCommand.CoordinateType OF 
// 'C R 010 MCS H +0250.00 +0000.00 +0500.00 +0000.00 +0045.00 +0180.00 BOR CLW H +0250.00 +0000.00 +0500.00 +0000.00 +0045.00 +0180.00'
	DUT_Command_CoordinateType.Literal:
		IF _CmdParams[12] = _PathChoiceClw THEN
			stCommand.PathChoice := MC_CIRC_PATHCHOICE.CLOCKWISE;
		ELSIF _CmdParams[12] = _PathChoiceCcw THEN
			stCommand.PathChoice := MC_CIRC_PATHCHOICE.COUNTER_CLOCKWISE;
		ELSE
			Error := TRUE;
			ErrorDescription := 'Incorrect circle direction';
		END_IF
		IF _CmdParams[13] = _CoordTypeH THEN
			stCommand.CircularCoordinateType := DUT_Command_CoordinateType.Literal;
		ELSIF _CmdParams[13] = _CoordTypeV THEN
			stCommand.CircularCoordinateType := DUT_Command_CoordinateType.Variable;
		ELSE
			Error := TRUE;
			ErrorDescription := 'Incorrect coordinate type'; // TODO yeah, this needs better naming. "coordinate type" does not fit.
		END_IF
// 'C R 010 MCS V S 001 BOR CLW H +0250.00 +0000.00 +0500.00 +0000.00 +0045.00 +0180.00'
	DUT_Command_CoordinateType.Variable:
		IF _CmdParams[8] = _PathChoiceClw THEN
			stCommand.PathChoice := MC_CIRC_PATHCHOICE.CLOCKWISE;
		ELSIF _CmdParams[8] = _PathChoiceCcw THEN
			stCommand.PathChoice := MC_CIRC_PATHCHOICE.COUNTER_CLOCKWISE;
		ELSE
			Error := TRUE;
			ErrorDescription := 'Incorrect circle direction';
		END_IF
		IF _CmdParams[9] = _CoordTypeH THEN
			stCommand.CircularCoordinateType := DUT_Command_CoordinateType.Literal;
		ELSIF _CmdParams[9] = _CoordTypeV THEN
			stCommand.CircularCoordinateType := DUT_Command_CoordinateType.Variable;
		ELSE
			Error := TRUE;
			ErrorDescription := 'Incorrect coordinate type'; // TODO this naming "coordinate type" needs to go.
		END_IF
	
END_CASE

//
CASE stCommand.CircularCoordinateType OF 
	DUT_Command_CoordinateType.Literal:
		CASE stCommand.CoordinateType OF
// 'C R 010 MCS H +0250.00 +0000.00 +0500.00 +0000.00 +0045.00 +0180.00 BOR CLW H +0250.00 +0000.00 +0500.00 +0000.00 +0045.00 +0180.00'
			DUT_Command_CoordinateType.Literal:
				stCommand.CoordRef2.X := STRING_TO_LREAL(_CmdParams[14]);
				stCommand.CoordRef2.Y := STRING_TO_LREAL(_CmdParams[15]);
				stCommand.CoordRef2.Z := STRING_TO_LREAL(_CmdParams[16]);
				stCommand.CoordRef2.A := STRING_TO_LREAL(_CmdParams[17]);
				stCommand.CoordRef2.B := STRING_TO_LREAL(_CmdParams[18]);
				stCommand.CoordRef2.C := STRING_TO_LREAL(_CmdParams[19]);
// 'C R 010 MCS V S 001 BOR CLW H +0250.00 +0000.00 +0500.00 +0000.00 +0045.00 +0180.00'
			DUT_Command_CoordinateType.Variable:
				stCommand.CoordRef2.X := STRING_TO_LREAL(_CmdParams[10]);
				stCommand.CoordRef2.Y := STRING_TO_LREAL(_CmdParams[11]);
				stCommand.CoordRef2.Z := STRING_TO_LREAL(_CmdParams[12]);
				stCommand.CoordRef2.A := STRING_TO_LREAL(_CmdParams[13]);
				stCommand.CoordRef2.B := STRING_TO_LREAL(_CmdParams[14]);
				stCommand.CoordRef2.C := STRING_TO_LREAL(_CmdParams[15]);
				
		END_CASE
	
	DUT_Command_CoordinateType.Variable:
		CASE stCommand.CoordinateType OF
// 'C R 010 MCS H +0250.00 +0000.00 +0500.00 +0000.00 +0045.00 +0180.00 BOR CLW V V 001'
			DUT_Command_CoordinateType.Literal:
				stCommand.CircularArrayIndex := STRING_TO_UINT(_CmdParams[15]);
				IF stCommand.CircularArrayIndex <= GVL.POS_ARR_END 
					AND stCommand.CircularArrayIndex >= GVL.POS_ARR_BEG THEN
						IF _CmdParams[14] = _ArrayTypeS THEN
							stCommand.CircularArrayType := DUT_Command_ArrayType.StoredPosition;
							stCommand.CoordRef2 := PersistentVars.StoredPositions[stCommand.CircularArrayIndex].Position;
						ELSIF _CmdParams[14] = _ArrayTypeV THEN
							stCommand.CircularArrayType := DUT_Command_ArrayType.VisionRegister;
							stCommand.CoordRef2 := PersistentVars.VisionRegisters[stCommand.CircularArrayIndex].Position;
						ELSE
							Error := TRUE;
							ErrorDescription := 'Incorrect array type';
						END_IF
					
				ELSE
					Error:=TRUE;
					ErrorDescription := 'Array index out of bounds';
					
				END_IF
				
// 'C R 010 MCS V S 001 BOR CLW V V 001'
			DUT_Command_CoordinateType.Variable:
				stCommand.CircularArrayIndex := STRING_TO_UINT(_CmdParams[11]);
				IF stCommand.CircularArrayIndex <= GVL.POS_ARR_END 
					AND stCommand.CircularArrayIndex >= GVL.POS_ARR_BEG THEN
						IF _CmdParams[10] = _ArrayTypeS THEN
							stCommand.CircularArrayType := DUT_Command_ArrayType.StoredPosition;
							stCommand.CoordRef2 := PersistentVars.StoredPositions[stCommand.CircularArrayIndex].Position;
						ELSIF _CmdParams[10] = _ArrayTypeV THEN
							stCommand.CircularArrayType := DUT_Command_ArrayType.VisionRegister;
							stCommand.CoordRef2 := PersistentVars.VisionRegisters[stCommand.CircularArrayIndex].Position;
						ELSE
							Error:=TRUE;
							ErrorDescription := 'Incorrect array type';
						END_IF
					
				ELSE
					Error:=TRUE;
					ErrorDescription := 'Array index out of bounds';
				END_IF
				
		END_CASE
	
END_CASE
                  
END_FUNCTION_BLOCK

PROGRAM _20_Io
VAR
	PowerOn: BOOL;
	
	Execute_Servo1: BOOL;
	Speed_Servo1: LREAL := 360;
	Position_Servo1: LREAL := 0;
	MC_Power_Servo1: MC_Power;
	MC_MoveAbsolute_Servo1: MC_MoveAbsolute;
END_VAR

                    //
PowerOn := GVL.PowerOn;

//
A_CmdIoMapping();

// servo 1
MC_Power_Servo1(
	Axis:= AdafruitPwm01, 
	Enable:= PowerOn, 
	bRegulatorOn:= PowerOn, 
	bDriveStart:= PowerOn, 
	Status=> , 
	bRegulatorRealState=> , 
	bDriveStartRealState=> , 
	Busy=> , 
	Error=> , 
	ErrorID=> );
	
MC_MoveAbsolute_Servo1(
	Axis:= AdafruitPwm01, 
	Execute:= Execute_Servo1, 
	Position:= Position_Servo1, 
	Velocity:= Speed_Servo1, 
	Acceleration:= 1000, 
	Deceleration:= 1000, 
	Jerk:= 1000, 
	Direction:= , 
	BufferMode:= , 
	Done=> , 
	Busy=> , 
	Active=> , 
	CommandAborted=> , 
	Error=> , 
	ErrorID=> );
Execute_Servo1 := FALSE;
                  

ACTION A_CmdIoMapping:
                        
//
GVL.CmdIO.Input := GVL.DigitalInput;
GVL.DigitalOutput := GVL.CmdIO.Output;

//
                      
END_ACTION
END_PROGRAM

PROGRAM _30_Visu
VAR	
	
	SelectedProgramNumber: INT;
	SelectedRecipeRowIndex: INT;
	RecipeRowSelected: BOOL;
	InsertLineAbove: BOOL;
	InsertLineBelow: BOOL;
	DeleteLine: BOOL;
	CopySelectedCommand: BOOL;
	CopiedCommandType: DUT_CommandType;
	CopiedCommandString: STRING(GVL.COMMAND_LEN);
	PasteCommand: BOOL;
	
	_i,_j,_k: INT;
	
	SetStoredPositionAsCurrent: BOOL;
	SelectedStoredPosition: UINT;
	SetVisionRegisterAsCurrent: BOOL;
	SelectedVisionRegister: UINT;
	SelectedFlag: UINT;
	
	//
	TeachPosition: BOOL;
	stTeachPosition: ST_MoveCmd;
	
	//
	MoveCmdParser: ParseMoveCmd;
	stMoveCmd: ST_MoveCmd;
	MoveCmdVisu: AddMoveCmd_VISU_STRUCT;
	
	//
	OutputCmdParser: ParseOutputCmd;
	stOutputCmd: ST_OutputCmd;
	OutputCmdVisu: AddOutputCmd_VISU_STRUCT;
	
	//
	PauseCmdParser: ParsePauseCmd;
	stPauseCmd: ST_PauseCmd;
	PauseCmdVisu: AddPauseCmd_VISU_STRUCT;
	
	//
	VisionCmdParser : ParseVisionCmd;
	stVisionCmd : ST_VisionCmd;
	VisionCmdVisu: AddVisionCmd_VISU_STRUCT;
	
	//
	VarSetCmdParser : ParseVarSetCmd;
	stVarSetCmd : ST_VarSetCmd;
	VarSetCmdVisu: AddVarSetCmd_VISU_STRUCT;
	
	//
	CncCmdParser : ParseCncCmd;
	stCncCmd : ST_CncCmd;
	CncCmdVisu: AddCncCmd_VISU_STRUCT;
	
	//
	LogicCmdParser : ParseLogicCmd;
	stLogicCmd : ST_LogicCmd;
	LogicCmdVisu: AddLogicCmd_VISU_STRUCT;
	
	//
	CurrentVisu: STRING;
	OpenDialog: VU.FbOpenDialogExtended;

END_VAR

                    
//
IF (InsertLineAbove OR InsertLineBelow) AND RecipeRowSelected THEN
	//
	IF InsertLineAbove THEN
		InsertLineAbove := FALSE;
		_j := SelectedRecipeRowIndex + 1;
	ELSIF InsertLineBelow THEN
		InsertLineBelow := FALSE;
		_j := SelectedRecipeRowIndex + 2;
	END_IF
	//
	FOR _i := GVL.PROG_CMDS_ARR_END TO _j BY -1 DO
		// shift all data
		IF _i >= GVL.PROG_CMDS_ARR_BEG AND _i <= GVL.PROG_CMDS_ARR_END THEN // can never really bo too careful am I right?
			PersistentVars.Programs[SelectedProgramNumber].Commands[_i].CommandType := PersistentVars.Programs[SelectedProgramNumber].Commands[_i - 1].CommandType;
			PersistentVars.Programs[SelectedProgramNumber].Commands[_i].CommandString := PersistentVars.Programs[SelectedProgramNumber].Commands[_i - 1].CommandString;
		END_IF
	END_FOR
	//
	PersistentVars.Programs[SelectedProgramNumber].Commands[_j - 1].CommandType := DUT_CommandType.Disabled;
	PersistentVars.Programs[SelectedProgramNumber].Commands[_j - 1].CommandString := '';
END_IF

//
IF DeleteLine AND RecipeRowSelected THEN
	DeleteLine := FALSE;
	FOR _i := SelectedRecipeRowIndex TO GVL.PROG_CMDS_ARR_END - 1 BY 1 DO
		IF _i >= GVL.PROG_CMDS_ARR_BEG AND _i <= GVL.PROG_CMDS_ARR_END THEN // can never really bo too careful am I right?
			PersistentVars.Programs[SelectedProgramNumber].Commands[_i].CommandType := PersistentVars.Programs[SelectedProgramNumber].Commands[_i + 1].CommandType;
			PersistentVars.Programs[SelectedProgramNumber].Commands[_i].CommandString := PersistentVars.Programs[SelectedProgramNumber].Commands[_i + 1].CommandString;
		END_IF
	END_FOR
END_IF

//
IF SetStoredPositionAsCurrent THEN
	SetStoredPositionAsCurrent := FALSE;
	PersistentVars.StoredPositions[SelectedStoredPosition].Position.X := F_RoundLreal(_00_Main.ProcessJog.Position.v[0],2);
	PersistentVars.StoredPositions[SelectedStoredPosition].Position.Y := F_RoundLreal(_00_Main.ProcessJog.Position.v[1],2);
	PersistentVars.StoredPositions[SelectedStoredPosition].Position.Z := F_RoundLreal(_00_Main.ProcessJog.Position.v[2],2);
	PersistentVars.StoredPositions[SelectedStoredPosition].Position.A := F_RoundLreal(_00_Main.ProcessJog.Position.v[3],2);
	PersistentVars.StoredPositions[SelectedStoredPosition].Position.B := F_RoundLreal(_00_Main.ProcessJog.Position.v[4],2);
	PersistentVars.StoredPositions[SelectedStoredPosition].Position.C := F_RoundLreal(_00_Main.ProcessJog.Position.v[5],2);
END_IF

//
IF TeachPosition THEN
	TeachPosition := FALSE;
	//
	stTeachPosition.MoveType := DUT_Command_MoveType.DirectMove;
	stTeachPosition.Speed := 50;
	stTeachPosition.PositionType := DUT_Command_PositionType.AbsolutePosition;
	stTeachPosition.CoordSystem := _00_Main.ProcessJog.CoordSystem;
	stTeachPosition.CoordRef.X := F_RoundLreal(_00_Main.ProcessJog.Position.v[0],2);
	stTeachPosition.CoordRef.Y := F_RoundLreal(_00_Main.ProcessJog.Position.v[1],2);
	stTeachPosition.CoordRef.Z := F_RoundLreal(_00_Main.ProcessJog.Position.v[2],2);
	stTeachPosition.CoordRef.A := F_RoundLreal(_00_Main.ProcessJog.Position.v[3],2);
	stTeachPosition.CoordRef.B := F_RoundLreal(_00_Main.ProcessJog.Position.v[4],2);
	stTeachPosition.CoordRef.C := F_RoundLreal(_00_Main.ProcessJog.Position.v[5],2);
	PersistentVars.Programs[SelectedProgramNumber].Commands[SelectedRecipeRowIndex].CommandType := DUT_CommandType.MoveCommand;
	PersistentVars.Programs[SelectedProgramNumber].Commands[SelectedRecipeRowIndex].CommandString := BuildMoveCmd(stTeachPosition);
END_IF

//
IF PasteCommand THEN
	PasteCommand := FALSE;
	PersistentVars.Programs[SelectedProgramNumber].Commands[SelectedRecipeRowIndex].CommandType := CopiedCommandType;
	PersistentVars.Programs[SelectedProgramNumber].Commands[SelectedRecipeRowIndex].CommandString := CopiedCommandString;
END_IF

//
IF CopySelectedCommand THEN
	CopySelectedCommand := FALSE;
	
	//
	CopiedCommandType := PersistentVars.Programs[SelectedProgramNumber].Commands[SelectedRecipeRowIndex].CommandType;
	CopiedCommandString := PersistentVars.Programs[SelectedProgramNumber].Commands[SelectedRecipeRowIndex].CommandString;
	
	CASE PersistentVars.Programs[SelectedProgramNumber].Commands[SelectedRecipeRowIndex].CommandType OF
		DUT_CommandType.Disabled:
			//
			
		DUT_CommandType.MoveCommand:
			MoveCmdParser(Command := PersistentVars.Programs[SelectedProgramNumber].Commands[SelectedRecipeRowIndex].CommandString);
			stMoveCmd := MoveCmdParser.stCommand;
			
		DUT_CommandType.PauseCommand:
			PauseCmdParser(Command:=PersistentVars.Programs[SelectedProgramNumber].Commands[SelectedRecipeRowIndex].CommandString);
			stPauseCmd := PauseCmdParser.stCommand;
			
		DUT_CommandType.InputCommand:
			//
			
		DUT_CommandType.OutputCommand:
			OutputCmdParser(Command:=PersistentVars.Programs[SelectedProgramNumber].Commands[SelectedRecipeRowIndex].CommandString);
			stOutputCmd := OutputCmdParser.stCommand;
			
		DUT_CommandType.VisionCommand:
			VisionCmdParser(Command:=PersistentVars.Programs[SelectedProgramNumber].Commands[SelectedRecipeRowIndex].CommandString);
			stVisionCmd := VisionCmdParser.stCommand;
			
		DUT_CommandType.VarSetCommand:
			VarSetCmdParser(Command:=PersistentVars.Programs[SelectedProgramNumber].Commands[SelectedRecipeRowIndex].CommandString);
			stVarSetCmd := VarSetCmdParser.stCommand;
			
		DUT_CommandType.CncCommand:
			CncCmdParser(Command:=PersistentVars.Programs[SelectedProgramNumber].Commands[SelectedRecipeRowIndex].CommandString);
			stCncCmd := CncCmdParser.stCommand;
			
		DUT_CommandType.LogicCommand:
			LogicCmdParser(Command:=PersistentVars.Programs[SelectedProgramNumber].Commands[SelectedRecipeRowIndex].CommandString);
			stLogicCmd := LogicCmdParser.stCommand;
			
	END_CASE
	
END_IF

// should be called after CopySelectedCommand case statement
CurrentVisu := VisuElems.CurrentVisu;
OpenDialog(
	xExecute:= , 
	xDone=> , 
	xBusy=> , 
	xError=> , 
	itfClientFilter:= , 
	eError=> , 
	sDialogName:= , 
	xModal:= TRUE, // TRUE - visu in background cannot be used
	pTopLeftPosition:= , 
	itfDialogOpenedListener:= , 
	pbyDialogInterfaceData:= , 
	udiDialogInterfaceDataSize:= , 
	itfDialogCloseListener:= , 
	pbyTagForDialogClosed:= , 
	dwDialogFlags:= );
IF (OpenDialog.xExecute AND OpenDialog.xDone) 
	OR OpenDialog.xError 
	THEN
		OpenDialog.xExecute := FALSE;
END_IF
                  
END_PROGRAM

FUNCTION BuildOutputCmd : STRING(GVL.COMMAND_LEN)
VAR_INPUT
	stCommand: ST_OutputCmd;
END_VAR
VAR
    _Command: STRING(GVL.COMMAND_LEN);
END_VAR
VAR CONSTANT
	_Delimiter: STRING:=' ';
	_OutTypeDig: STRING(3):='DIG';
	_OutTypeAna: STRING(3):='ANA';
	_OutTypeSrv: STRING(3):='SRV';
END_VAR

                    // DIG +0001.00 +0001.00 (turn digital input 1 on)
// DIG +0001.00 +0000.00 (turn digital input 1 off)
// SRV +0001.00 +0030.00 +0360.00(set servo 1 to position 30 at speed 360)

// clear the command
_Command:='';

//
CASE stCommand.OutputType OF
	DUT_OutputType.Digital:
		F_AddElement(_Command, _Delimiter, _OutTypeDig);
	DUT_OutputType.Analog:
		F_AddElement(_Command, _Delimiter, _OutTypeAna);
	Dut_OutputType.Servo:
		F_AddElement(_Command, _Delimiter, _OutTypeSrv);
END_CASE

//
F_AddElement(_Command, _Delimiter, INT_TO_STRING(stCommand.OutputTarget));

//
F_AddElement(_Command, _Delimiter, LREAL_TO_STRING(stCommand.OutputValue1));

// only need if servo
IF stCommand.OutputType = DUT_OutputType.Servo THEN
	F_AddElement(_Command, _Delimiter, LREAL_TO_STRING(stCommand.OutputValue2));
END_IF

// set function equal to command
BuildOutputCmd := _Command;
                  
END_FUNCTION

FUNCTION_BLOCK ParseOutputCmd
VAR_INPUT
	Command: STRING(GVL.COMMAND_LEN);
END_VAR
VAR_OUTPUT
	stCommand: ST_OutputCmd;
	Error: BOOL;
	ErrorDescription: STRING;
END_VAR
VAR
	_CmdParams: ARRAY [0..GVL.COMMAND_LEN] OF STRING;
	_OutputType: STRING;
END_VAR

                    // DIG 1 1 (turn digital input 1 on)
// DIG 1 0 (turn digital input 1 off)
// SRV 1 30.0 360.0(set servo 1 to position 30 at speed 360)

Error:=FALSE;
ErrorDescription:='';

// split command string into commands
_CmdParams:=F_SplitCmd(Command:=Command);

_OutputType := _CmdParams[0];
IF _OutputType = 'DIG' THEN
	stCommand.OutputType := DUT_OutputType.Digital;
ELSIF _OutputType = 'ANA' THEN
	stCommand.OutputType := DUT_OutputType.Analog;
ELSIF _OutputType = 'SRV' THEN
	stCommand.OutputType := DUT_OutputType.Servo;
END_IF
stCommand.OutputTarget := STRING_TO_INT(_CmdParams[1]);
stCommand.OutputValue1 := STRING_TO_LREAL(_CmdParams[2]);

// only need to parse the second parameter if not digital
IF NOT (stCommand.OutputType = DUT_OutputType.Digital) THEN
	stCommand.OutputValue2 := STRING_TO_LREAL(_CmdParams[3]);
END_IF
                  
END_FUNCTION_BLOCK

FUNCTION BuildPauseCmd : STRING(GVL.COMMAND_LEN)
VAR_INPUT
	stCommand: ST_PauseCmd;
END_VAR
VAR
    _Command: STRING(GVL.COMMAND_LEN);
END_VAR
VAR CONSTANT
	_Delimiter: STRING:=' ';
END_VAR

                    // clear the command
_Command:='';

// build command
F_AddElement(_Command, _Delimiter, TIME_TO_STRING(stCommand.PauseTime));

// set function equal to command
BuildPauseCmd := _Command;
                  
END_FUNCTION

FUNCTION_BLOCK ParsePauseCmd
VAR_INPUT
	Command: STRING(GVL.COMMAND_LEN);
END_VAR
VAR_OUTPUT
	stCommand: ST_PauseCmd;
	Error: BOOL;
	ErrorDescription: STRING;
END_VAR
VAR
	_CmdParams: ARRAY [0..GVL.COMMAND_LEN] OF STRING;
END_VAR

                    // T#30s

Error:=FALSE;
ErrorDescription:='';

// split command string into commands
_CmdParams:=F_SplitCmd(Command:=Command);

stCommand.PauseTime := STRING_TO_TIME(_CmdParams[0]);
                  
END_FUNCTION_BLOCK

PROGRAM _40_Vision
VAR
	ProcessVisionCommand: VisionCmdProcessor;
END_VAR

                    //
ProcessVisionCommand(
	StoredPositions:= PersistentVars.StoredPositions,
	VisionRegisters:= PersistentVars.VisionRegisters,
	Flags:= PersistentVars.Flags,
	ItfUnitMode=> ,
	Error=> , 
	ErrorDescription=> , 
	VisionStateText=> );
                  
END_PROGRAM

FUNCTION_BLOCK CncPathPlanner
VAR_IN_OUT
	VarList: SMC_VarList;
END_VAR
VAR_INPUT
END_VAR
VAR_OUTPUT
	DataOut: POINTER TO SMC_OUTQUEUE;
	Busy: BOOL;
	Done: BOOL;
	Error: BOOL;
	ErrorDescription: STRING;
END_VAR
VAR
	_Filename: STRING := '_cnc/CNC_FromFile.cnc';
	_SMC_NCInterpreter: SMC_NCInterpreter;
	_SMC_ReadNCFile2: SMC_ReadNCFile2;
	_SMC_CheckVelocities: SMC_CheckVelocities;
	_SMC_GEOINFO: ARRAY[0..49] OF SMC_GEOINFO;
	_StartPos: SMC_PosInfo;
	_OriConvention: SMC_ORI_CONVENTION := SMC_ORI_CONVENTION.XYZ;
	_ExecuteRtrig: R_TRIG;
	_Execute: BOOL;
	_ResetRtrig: R_TRIG;
	_Reset: BOOL;
	_Sequence: INT:=0;
	_ErrorRtrig: R_TRIG;
END_VAR
VAR CONSTANT
	_BaseCncDirectory: STRING:='_cnc/'; // before update to 3.5.19.40 '/var/opt/codesys/_cnc/'
END_VAR

                    _ExecuteRtrig(CLK:=_Execute);
IF _ExecuteRtrig.Q THEN
	_Execute:= FALSE;
END_IF
_ResetRtrig(CLK:=_Reset);
IF _ResetRtrig.Q THEN
	_Reset:= FALSE;
	_Sequence:=999;
END_IF

Busy := _Sequence <> 000;

CASE _Sequence OF
	999:
		_SMC_ReadNCFile2.bExecute := FALSE;
		_Sequence := 000;
	000:
		IF _ExecuteRtrig.Q THEN
			_SMC_ReadNCFile2.bExecute := TRUE;
			_Sequence := 1;
		END_IF
	001:
		IF NOT _SMC_CheckVelocities.bBusy THEN
			_Sequence := 999;
			Done := TRUE;
		END_IF
	
END_CASE

_SMC_ReadNCFile2(
	bExecute:= , 
	bAbort:= _Sequence = 999, 
	sFileName:= _Filename, 
	pvl:= ADR(VarList), 
	fDefaultVel:= , 
	fDefaultAccel:= , 
	fDefaultDecel:= , 
	fDefaultVelFF:= , 
	fDefaultAccelFF:= , 
	fDefaultDecelFF:= , 
	b3DMode:= , 
	bStepSuppress:= , 
	aSubProgramDirs:= , 
	bParenthesesAsComments:= , 
	bDisableJumpBuffer:= , 
	pCustomFunTable:= , 
	aTokenModifier:= , 
	aSentenceModifier:= , 
	bBusy=> , 
	bError=> , 
	ErrorID=> , 
	errorPos=> , 
	ErrorProgramName=> , 
	sentences=> , 
	adwFileSize=> , 
	adwPos=> );

_SMC_NCInterpreter(
	sentences:= _SMC_ReadNCFile2.sentences, 
	bExecute:= _SMC_ReadNCFile2.bExecute, 
	bAbort:= _Sequence = 999, 
	bAppend:= , 
	piStartPosition:= _StartPos, 
	vStartToolLength:= , 
	nSizeOutQueue:= SIZEOF(_SMC_GEOINFO), 
	pbyBufferOutQueue:= ADR(_SMC_GEOINFO), 
	bEnableSyntaxChecks:= , 
	eOriConv:= _OriConvention, // SMC_ORI_CONVENTION 
	dCircleTolerance:= , 
	pInterpreterStack:= , 
	nInterpreterStackSizeBytes:= , 
	bDone=> , 
	bBusy=> , 
	bError=> , 
	wErrorID=> , 
	errorPos=> , 
	poqDataOut=> , 
	iStatus=> , 
	iLineNumberDecoded=> , 
	GCodeText=> , 
	CallstackInfo=> , 
	aActivePrograms=> );

_SMC_CheckVelocities(
	bExecute:= _SMC_NCInterpreter.bExecute, 
	bAbort:= _Sequence = 999, 
	poqDataIn:= _SMC_NCInterpreter.poqDataOut, 
	dAngleTol:= , 
	bCheckAddAxVelJump:= , 
	dMaxAddAxVelDifference:= , 
	bBusy=> , 
	bError=> , 
	wErrorID=> , 
	poqDataOut=> DataOut);
	
_ErrorRtrig();
_ErrorRtrig.CLK:= _SMC_ReadNCFile2.bError
				OR _SMC_NCInterpreter.bError
				OR _SMC_CheckVelocities.bError;
IF _ErrorRtrig.Q THEN
	Error := TRUE;
	IF _SMC_ReadNCFile2.bError THEN
		ErrorDescription := CONCAT('ReadNCFile Error: ',
                                CONCAT(TO_STRING(_SMC_ReadNCFile2.ErrorID),
                                CONCAT(' ', SMC_ErrorString(_SMC_ReadNCFile2.ErrorID,
                                            SMC_Language_Type.english)))) ;
	END_IF
	IF _SMC_NCInterpreter.bError THEN
		ErrorDescription := CONCAT(' NCInterpreter Error: ',
                                CONCAT(TO_STRING(_SMC_NCInterpreter.wErrorID),
                                CONCAT(' ', SMC_ErrorString(_SMC_NCInterpreter.wErrorID,
                                            SMC_Language_Type.english)))) ;
	END_IF
	IF _SMC_CheckVelocities.bError THEN
		ErrorDescription := CONCAT(' CheckVelocities Error: ',
                                CONCAT(TO_STRING(_SMC_CheckVelocities.wErrorID),
                                CONCAT(' ', SMC_ErrorString(_SMC_CheckVelocities.wErrorID,
                                            SMC_Language_Type.english)))) ;
	END_IF
END_IF
                  

METHOD PUBLIC M_Execute : BOOL
VAR_INPUT
	Filename: STRING := 'CNC_FromFile.cnc';
END_VAR
                          _Filename := CONCAT(_BaseCncDirectory, Filename);
_Execute:=TRUE;
Done := FALSE;
                        
END_METHOD

METHOD PUBLIC M_Reset : BOOL
VAR_INPUT
END_VAR
                          _Reset := TRUE;
Error := FALSE;
ErrorDescription := '';
                        
END_METHOD

METHOD PUBLIC M_SetStartPosition : BOOL
VAR_INPUT
	StartPos: SMC_PosInfo;
END_VAR
                          _StartPos := StartPos;
                        
END_METHOD

METHOD PUBLIC M_SetOriConvention : BOOL
VAR_INPUT
	OriConvention: SMC_ORI_CONVENTION := SMC_ORI_CONVENTION.XYZ;
END_VAR
                          _OriConvention := OriConvention;
                        
END_METHOD
END_FUNCTION_BLOCK

FUNCTION BuildCncCmd : STRING(GVL.COMMAND_LEN)
VAR_INPUT
	stCommand: ST_CncCmd;
END_VAR
VAR
	_Command: STRING(GVL.COMMAND_LEN);
END_VAR
VAR CONSTANT
	_Delimiter: STRING:=' ';
	_AddString: STRING(3):='ADD';
	_XYZString: STRING(3):='XYZ';
	_ZYXString: STRING(3):='ZYX';
	_ZYZString: STRING(3):='ZYZ';
	_LiteralString: STRING(3):='LIT';
	_VariableString: STRING(3):='VAR';
	_StoredPositionsString: STRING(3):='STO';
	_VisionRegistersString: STRING(3):='VIS';
	_FlagsString: STRING(3):='FLG';
END_VAR

                    // /path/to/file/with/no/spaces/file.cnc ADD|XYX|ZYX|ZYZ startpos
// file1.cnc XYZ H +0250.00 +0000.00 +0500.00 +0000.00 +0045.00 +0180.00
// file2.cnc ADD A S 025
// file3.cnc ADD A V 015

_Command:='';

//
F_AddElement(_Command, _Delimiter, stCommand.Filename);

//
CASE stCommand.OriConvention OF
	SMC_ORI_CONVENTION.ADDAXES:
		F_AddElement(_Command, _Delimiter, _AddString);
	SMC_ORI_CONVENTION.XYZ:
		F_AddElement(_Command, _Delimiter, _XYZString);
	SMC_ORI_CONVENTION.ZYX:
		F_AddElement(_Command, _Delimiter, _ZYXString);
	SMC_ORI_CONVENTION.ZYZ:
		F_AddElement(_Command, _Delimiter, _ZYZString);
END_CASE

//
CASE stCommand.CoordinateType OF
	DUT_Command_CoordinateType.Literal:
		F_AddElement(_Command, _Delimiter, _LiteralString);
		F_AddElement(_Command, _Delimiter, LREAL_TO_STRING(stCommand.StartPos.dX));
		F_AddElement(_Command, _Delimiter, LREAL_TO_STRING(stCommand.StartPos.dY));
		F_AddElement(_Command, _Delimiter, LREAL_TO_STRING(stCommand.StartPos.dZ));
		F_AddElement(_Command, _Delimiter, LREAL_TO_STRING(stCommand.StartPos.dA));
		F_AddElement(_Command, _Delimiter, LREAL_TO_STRING(stCommand.StartPos.dB));
		F_AddElement(_Command, _Delimiter, LREAL_TO_STRING(stCommand.StartPos.dC));
		
	DUT_Command_CoordinateType.Variable:
		F_AddElement(_Command, _Delimiter, _VariableString);
		CASE stCommand.ArrayType OF
			DUT_Command_ArrayType.StoredPosition:
				F_AddElement(_Command, _Delimiter, _StoredPositionsString);
			DUT_Command_ArrayType.VisionRegister:
				F_AddElement(_Command, _Delimiter, _VisionRegistersString);
			DUT_Command_ArrayType.Flag:
				F_AddElement(_Command, _Delimiter, _FlagsString);
		END_CASE
		F_AddElement(_Command, _Delimiter, INT_TO_STRING(stCommand.ArrayIndex));
		
END_CASE

BuildCncCmd := _Command;

                  
END_FUNCTION

FUNCTION_BLOCK PositionTracker
VAR_IN_OUT
	AxisGroup: AXIS_GROUP_REF_SM3;
	SM3_Drive_PosControl_J1: SM3_Drive_PosControl.AXIS_REF_POSCONTROL;
	SM3_Drive_PosControl_J2: SM3_Drive_PosControl.AXIS_REF_POSCONTROL;
	SM3_Drive_PosControl_J3: SM3_Drive_PosControl.AXIS_REF_POSCONTROL;
	SM3_Drive_PosControl_J4: SM3_Drive_PosControl.AXIS_REF_POSCONTROL;
	SM3_Drive_PosControl_J5: SM3_Drive_PosControl.AXIS_REF_POSCONTROL;
	SM3_Drive_PosControl_J6: SM3_Drive_PosControl.AXIS_REF_POSCONTROL;
END_VAR
VAR_INPUT
END_VAR
VAR_OUTPUT
	VisuStruct3DTrack: VisuStruct3DTrack;
	Arm: SMC_ArticulatedRobot_6DOF_J0_State;
	Elbow: SMC_ArticulatedRobot_6DOF_J1_State;
	Hand: SMC_ArticulatedRobot_6DOF_J4_State;
END_VAR
VAR
	_SMC_Trafof_ArticulatedRobot_6DOF: SMC_Trafof_ArticulatedRobot_6DOF;
	_SMC_TrafoConfig_ArticulatedRobot_6DOF: SMC_TrafoConfig_ArticulatedRobot_6DOF;
	_VisuStruct3DPathPoint: ARRAY [0..10000] OF VisuStruct3DPathPoint;
	_SMC_PositionTracker: SMC_PositionTracker;
	_PositionTrackerClearR_Trig: R_Trig;
	_Clear: BOOL:=FALSE;
END_VAR

                    
// NOTE currently the settings for J6 invert direction under scaling/mapping contradict using motion control 
// libraries and CNC. For CNC to work properly, the setting is required to be enabled (inverted). Additionally
// the homing direction and position will need to be negated. This all requires a full download. Will be leaving 
// setting disabled for now so that we can continue to use motion control. 
//
// to recap, take these steps if you would like to try out CNC:
// 1. open the axis pool settings and under the scaling/mapping section enable 'invert direction'
// 2. in the A_Homing POU, change the homing direction to positive.
// 3. in _00_MAIN POU, under FirstScan set the initial home offset to a positive value (keep the value and just change the sign).
// 4. do a full download.
// 5. go online and set the persistent value (if previously initialized in FirstScan) to a positive value.
//
// UPDATE: Figured out a work around for this issue. In the A_Interpolater POU, I negated the set position in the ControlAxisByPos
// function block for J6 such that it drives the opposite way. This appears to have resolved the issue. Why this is needed, I do not
// know. I am sure it is some minor overlooked detail somewhere in the code...


_SMC_TrafoConfig_ArticulatedRobot_6DOF.a1:=ArfBotAxisGroup.Trafo.a1;//AxisGroup.Trafo.a1;
_SMC_TrafoConfig_ArticulatedRobot_6DOF.a2:=ArfBotAxisGroup.Trafo.a2;//AxisGroup.Trafo.a2;
_SMC_TrafoConfig_ArticulatedRobot_6DOF.a3:=ArfBotAxisGroup.Trafo.a3;//AxisGroup.Trafo.a3;
// conflicting documentation on if d1 needs to be pos or neg. only works as negative otherwise trafo reports invalid configuration
// https://product-help.schneider-electric.com/Machine%20Expert/V2.0/zh/codesys_softmotion/codesys_softmotion/modules/_sm_trafo_pou_six_dof_robot.html
// https://forge.codesys.com/forge/talk/Motion/thread/16e1f0327f/
_SMC_TrafoConfig_ArticulatedRobot_6DOF.d1:=-ArfBotAxisGroup.Trafo.d1;//-AxisGroup.Trafo.d1;
_SMC_TrafoConfig_ArticulatedRobot_6DOF.d3:=ArfBotAxisGroup.Trafo.d3;//AxisGroup.Trafo.d3;
_SMC_TrafoConfig_ArticulatedRobot_6DOF.d4:=ArfBotAxisGroup.Trafo.d4;//AxisGroup.Trafo.d4;
_SMC_TrafoConfig_ArticulatedRobot_6DOF.d6:=ArfBotAxisGroup.Trafo.d6;//AxisGroup.Trafo.d6;
_SMC_TrafoConfig_ArticulatedRobot_6DOF.q3_max_deg:=160; // TODO put magic numbers somewhere appropriate
_SMC_TrafoConfig_ArticulatedRobot_6DOF.q3_min_deg:=-160; // TODO put magic numbers somewhere appropriate
_SMC_TrafoConfig_ArticulatedRobot_6DOF.q5_max_deg:=160; // TODO put magic numbers somewhere appropriate
_SMC_TrafoConfig_ArticulatedRobot_6DOF.q5_min_deg:=-160; // TODO put magic numbers somewhere appropriate

// track position
_SMC_Trafof_ArticulatedRobot_6DOF(config:=_SMC_TrafoConfig_ArticulatedRobot_6DOF,
							Drive0:=SM3_Drive_PosControl_J1,
							Drive1:=SM3_Drive_PosControl_J2,
							Drive2:=SM3_Drive_PosControl_J3,
							Drive3:=SM3_Drive_PosControl_J4,
							Drive4:=SM3_Drive_PosControl_J5,
							Drive5:=SM3_Drive_PosControl_J6,
							vToolPos=>,
							mToolOrientation=>,
							armState=>Arm,
							elbowState=>Elbow,
							handState=>Hand);

_PositionTrackerClearR_Trig(Clk:=_Clear);
_SMC_PositionTracker(
	bEnable:= TRUE, 
	bClear:= _PositionTrackerClearR_Trig.Q, 
	dX:= _SMC_Trafof_ArticulatedRobot_6DOF.vToolPos.dX, 
	dY:= _SMC_Trafof_ArticulatedRobot_6DOF.vToolPos.dY, 
	dZ:= _SMC_Trafof_ArticulatedRobot_6DOF.vToolPos.dZ, 
	udiNumberOfPointsInArray:= 10001, //SIZEOF(_VisuStruct3DPathPoint), TODO make this dynamic. hint SIZEOF wont work
	pBuffer:= ADR(_VisuStruct3DPathPoint), 
	vs3dt=> VisuStruct3DTrack);
_Clear := FALSE;
                  

METHOD PUBLIC M_Clear
VAR_INPUT
END_VAR
                          _Clear := TRUE;
                        
END_METHOD
END_FUNCTION_BLOCK

FUNCTION_BLOCK OpenCV
VAR_INPUT
	sIpAddress: STRING(19):='127.0.0.1';
	uPort: UINT:=50011;
END_VAR
VAR_OUTPUT
END_VAR
VAR
	_Done: BOOL;
	_Busy: BOOL;
	_Error: BOOL;
	_ErrorDescription: STRING;
	_Response: STRING(255);
	_WorkerUid: STRING;
	_Execute: BOOL;
	_Reset: BOOL:=FALSE;
	_ResetRtrig: R_TRIG;
	_Step: INT;
	_Command: STRING(255);
	_ReadRecordLast: DINT;
	_PythonTcpClient: PythonTcpClient;
	_TimeoutTimer: TON:=(PT:=T#120S);
END_VAR

